    (* Table initialization: fTable_C *)
    fTable_C[0, 0] := 10.0000; fTable_C[0, 1] := -9999; fTable_C[0, 2] := 0.806885;
    fTable_C[1, 0] := 10.1617; fTable_C[1, 1] := -9999; fTable_C[1, 2] := 0.851522;
    fTable_C[2, 0] := 10.3261; fTable_C[2, 1] := -9999; fTable_C[2, 2] := 0.898628;
    fTable_C[3, 0] := 10.4931; fTable_C[3, 1] := -9999; fTable_C[3, 2] := 0.948341;
    fTable_C[4, 0] := 10.6628; fTable_C[4, 1] := -9999; fTable_C[4, 2] := 1.00080;
    fTable_C[5, 0] := 10.8353; fTable_C[5, 1] := -9999; fTable_C[5, 2] := 1.05755;
    fTable_C[6, 0] := 11.0106; fTable_C[6, 1] := -9999; fTable_C[6, 2] := 1.12167;
    fTable_C[7, 0] := 11.1886; fTable_C[7, 1] := -9999; fTable_C[7, 2] := 1.18968;
    fTable_C[8, 0] := 11.3696; fTable_C[8, 1] := -9999; fTable_C[8, 2] := 1.26181;
    fTable_C[9, 0] := 11.5535; fTable_C[9, 1] := -9999; fTable_C[9, 2] := 1.33832;
    fTable_C[10, 0] := 11.7404; fTable_C[10, 1] := -9999; fTable_C[10, 2] := 1.41946;
    fTable_C[11, 0] := 11.9303; fTable_C[11, 1] := -9999; fTable_C[11, 2] := 1.50553;
    fTable_C[12, 0] := 12.1232; fTable_C[12, 1] := -9999; fTable_C[12, 2] := 1.58971;
    fTable_C[13, 0] := 12.3193; fTable_C[13, 1] := -9999; fTable_C[13, 2] := 1.67820;
    fTable_C[14, 0] := 12.5186; fTable_C[14, 1] := -9999; fTable_C[14, 2] := 1.77161;
    fTable_C[15, 0] := 12.7210; fTable_C[15, 1] := -9999; fTable_C[15, 2] := 1.87023;
    fTable_C[16, 0] := 12.9268; fTable_C[16, 1] := -9999; fTable_C[16, 2] := 1.97433;
    fTable_C[17, 0] := 13.1359; fTable_C[17, 1] := -9999; fTable_C[17, 2] := 2.08423;
    fTable_C[18, 0] := 13.3483; fTable_C[18, 1] := -9999; fTable_C[18, 2] := 2.20025;
    fTable_C[19, 0] := 13.5642; fTable_C[19, 1] := -9999; fTable_C[19, 2] := 2.29235;
    fTable_C[20, 0] := 13.7836; fTable_C[20, 1] := -9999; fTable_C[20, 2] := 2.38287;
    fTable_C[21, 0] := 14.0066; fTable_C[21, 1] := -9999; fTable_C[21, 2] := 2.47696;
    fTable_C[22, 0] := 14.2331; fTable_C[22, 1] := -9999; fTable_C[22, 2] := 2.57477;
    fTable_C[23, 0] := 14.4633; fTable_C[23, 1] := -9999; fTable_C[23, 2] := 2.67645;
    fTable_C[24, 0] := 14.6973; fTable_C[24, 1] := -9999; fTable_C[24, 2] := 2.77114;
    fTable_C[25, 0] := 14.9350; fTable_C[25, 1] := -9999; fTable_C[25, 2] := 2.84605;
    fTable_C[26, 0] := 15.1765; fTable_C[26, 1] := -9999; fTable_C[26, 2] := 2.92298;
    fTable_C[27, 0] := 15.4220; fTable_C[27, 1] := -9999; fTable_C[27, 2] := 3.00199;
    fTable_C[28, 0] := 15.6714; fTable_C[28, 1] := -9999; fTable_C[28, 2] := 3.08313;
    fTable_C[29, 0] := 15.9249; fTable_C[29, 1] := -9999; fTable_C[29, 2] := 3.16647;
    fTable_C[30, 0] := 16.1825; fTable_C[30, 1] := -9999; fTable_C[30, 2] := 3.24213;
    fTable_C[31, 0] := 16.4442; fTable_C[31, 1] := -9999; fTable_C[31, 2] := 3.28778;
    fTable_C[32, 0] := 16.7102; fTable_C[32, 1] := -9999; fTable_C[32, 2] := 3.33408;
    fTable_C[33, 0] := 16.9805; fTable_C[33, 1] := -9999; fTable_C[33, 2] := 3.38103;
    fTable_C[34, 0] := 17.2551; fTable_C[34, 1] := -9999; fTable_C[34, 2] := 3.42863;
    fTable_C[35, 0] := 17.5342; fTable_C[35, 1] := -9999; fTable_C[35, 2] := 3.47691;
    fTable_C[36, 0] := 17.8178; fTable_C[36, 1] := -9999; fTable_C[36, 2] := 3.52041;
    fTable_C[37, 0] := 18.1060; fTable_C[37, 1] := -9999; fTable_C[37, 2] := 3.54277;
    fTable_C[38, 0] := 18.3989; fTable_C[38, 1] := -9999; fTable_C[38, 2] := 3.56528;
    fTable_C[39, 0] := 18.6964; fTable_C[39, 1] := -9999; fTable_C[39, 2] := 3.58793;
    fTable_C[40, 0] := 18.9988; fTable_C[40, 1] := -9999; fTable_C[40, 2] := 3.61072;
    fTable_C[41, 0] := 19.3061; fTable_C[41, 1] := -9999; fTable_C[41, 2] := 3.63366;
    fTable_C[42, 0] := 19.6184; fTable_C[42, 1] := -9999; fTable_C[42, 2] := 3.65674;
    fTable_C[43, 0] := 19.9357; fTable_C[43, 1] := -9999; fTable_C[43, 2] := 3.67997;
    fTable_C[44, 0] := 20.2582; fTable_C[44, 1] := -9999; fTable_C[44, 2] := 3.70335;
    fTable_C[45, 0] := 20.5858; fTable_C[45, 1] := -9999; fTable_C[45, 2] := 3.69489;
    fTable_C[46, 0] := 20.9188; fTable_C[46, 1] := -9999; fTable_C[46, 2] := 3.67204;
    fTable_C[47, 0] := 21.2571; fTable_C[47, 1] := -9999; fTable_C[47, 2] := 3.64934;
    fTable_C[48, 0] := 21.6009; fTable_C[48, 1] := -9999; fTable_C[48, 2] := 3.62677;
    fTable_C[49, 0] := 21.9503; fTable_C[49, 1] := -9999; fTable_C[49, 2] := 3.60434;
    fTable_C[50, 0] := 22.3053; fTable_C[50, 1] := -9999; fTable_C[50, 2] := 3.58205;
    fTable_C[51, 0] := 22.6661; fTable_C[51, 1] := -9999; fTable_C[51, 2] := 3.55990;
    fTable_C[52, 0] := 23.0327; fTable_C[52, 1] := -9999; fTable_C[52, 2] := 3.53320;
    fTable_C[53, 0] := 23.4053; fTable_C[53, 1] := -9999; fTable_C[53, 2] := 3.47892;
    fTable_C[54, 0] := 23.7838; fTable_C[54, 1] := -9999; fTable_C[54, 2] := 3.42547;
    fTable_C[55, 0] := 24.1685; fTable_C[55, 1] := -9999; fTable_C[55, 2] := 3.37285;
    fTable_C[56, 0] := 24.5594; fTable_C[56, 1] := -9999; fTable_C[56, 2] := 3.32103;
    fTable_C[57, 0] := 24.9566; fTable_C[57, 1] := -9999; fTable_C[57, 2] := 3.27000;
    fTable_C[58, 0] := 25.3603; fTable_C[58, 1] := -9999; fTable_C[58, 2] := 3.21977;
    fTable_C[59, 0] := 25.7705; fTable_C[59, 1] := -9999; fTable_C[59, 2] := 3.17030;
    fTable_C[60, 0] := 26.1873; fTable_C[60, 1] := -9999; fTable_C[60, 2] := 3.12096;
    fTable_C[61, 0] := 26.6109; fTable_C[61, 1] := -9999; fTable_C[61, 2] := 3.06350;
    fTable_C[62, 0] := 27.0413; fTable_C[62, 1] := -9999; fTable_C[62, 2] := 3.00708;
    fTable_C[63, 0] := 27.4786; fTable_C[63, 1] := -9999; fTable_C[63, 2] := 2.95171;
    fTable_C[64, 0] := 27.9231; fTable_C[64, 1] := -9999; fTable_C[64, 2] := 2.89736;
    fTable_C[65, 0] := 28.3747; fTable_C[65, 1] := -9999; fTable_C[65, 2] := 2.84401;
    fTable_C[66, 0] := 28.8337; fTable_C[66, 1] := -9999; fTable_C[66, 2] := 2.79164;
    fTable_C[67, 0] := 29.3000; fTable_C[67, 1] := 3.63318; fTable_C[67, 2] := 2.74024;
    fTable_C[68, 0] := 29.7739; fTable_C[68, 1] := 3.67378; fTable_C[68, 2] := 2.68978;
    fTable_C[69, 0] := 30.2555; fTable_C[69, 1] := 3.71270; fTable_C[69, 2] := 2.63618;
    fTable_C[70, 0] := 30.7449; fTable_C[70, 1] := 3.74753; fTable_C[70, 2] := 2.58360;
    fTable_C[71, 0] := 31.2421; fTable_C[71, 1] := 3.77973; fTable_C[71, 2] := 2.53206;
    fTable_C[72, 0] := 31.7475; fTable_C[72, 1] := 3.80969; fTable_C[72, 2] := 2.48155;
    fTable_C[73, 0] := 32.2609; fTable_C[73, 1] := 3.83764; fTable_C[73, 2] := 2.43205;
    fTable_C[74, 0] := 32.7827; fTable_C[74, 1] := 3.86374; fTable_C[74, 2] := 2.38354;
    fTable_C[75, 0] := 33.3130; fTable_C[75, 1] := 3.88807; fTable_C[75, 2] := 2.33599;
    fTable_C[76, 0] := 33.8518; fTable_C[76, 1] := 3.91071; fTable_C[76, 2] := 2.28940;
    fTable_C[77, 0] := 34.3993; fTable_C[77, 1] := 3.93156; fTable_C[77, 2] := 2.24373;
    fTable_C[78, 0] := 34.9557; fTable_C[78, 1] := 3.95026; fTable_C[78, 2] := 2.19898;
    fTable_C[79, 0] := 35.5211; fTable_C[79, 1] := 3.96709; fTable_C[79, 2] := 2.15799;
    fTable_C[80, 0] := 36.0956; fTable_C[80, 1] := 3.98488; fTable_C[80, 2] := 2.11827;
    fTable_C[81, 0] := 36.6794; fTable_C[81, 1] := 4.00253; fTable_C[81, 2] := 2.07928;
    fTable_C[82, 0] := 37.2727; fTable_C[82, 1] := 4.01992; fTable_C[82, 2] := 2.04101;
    fTable_C[83, 0] := 37.8755; fTable_C[83, 1] := 4.03712; fTable_C[83, 2] := 2.00344;
    fTable_C[84, 0] := 38.4882; fTable_C[84, 1] := 4.05432; fTable_C[84, 2] := 1.96657;
    fTable_C[85, 0] := 39.1107; fTable_C[85, 1] := 4.07360; fTable_C[85, 2] := 1.93037;
    fTable_C[86, 0] := 39.7432; fTable_C[86, 1] := 4.09449; fTable_C[86, 2] := 1.89011;
    fTable_C[87, 0] := 40.3861; fTable_C[87, 1] := 4.11010; fTable_C[87, 2] := 1.84650;
    fTable_C[88, 0] := 41.0393; fTable_C[88, 1] := 4.12229; fTable_C[88, 2] := 1.80390;
    fTable_C[89, 0] := 41.7031; fTable_C[89, 1] := 4.13211; fTable_C[89, 2] := 1.76228;
    fTable_C[90, 0] := 42.3776; fTable_C[90, 1] := 4.13985; fTable_C[90, 2] := 1.72163;
    fTable_C[91, 0] := 43.0630; fTable_C[91, 1] := 4.14559; fTable_C[91, 2] := 1.68191;
    fTable_C[92, 0] := 43.7595; fTable_C[92, 1] := 4.14925; fTable_C[92, 2] := 1.64310;
    fTable_C[93, 0] := 44.4673; fTable_C[93, 1] := 4.14955; fTable_C[93, 2] := 1.60520;
    fTable_C[94, 0] := 45.1865; fTable_C[94, 1] := 4.14584; fTable_C[94, 2] := 1.56917;
    fTable_C[95, 0] := 45.9174; fTable_C[95, 1] := 4.14175; fTable_C[95, 2] := 1.54376;
    fTable_C[96, 0] := 46.6600; fTable_C[96, 1] := 4.14174; fTable_C[96, 2] := 1.51876;
    fTable_C[97, 0] := 47.4147; fTable_C[97, 1] := 4.14300; fTable_C[97, 2] := 1.49417;
    fTable_C[98, 0] := 48.1816; fTable_C[98, 1] := 4.14486; fTable_C[98, 2] := 1.46998;
    fTable_C[99, 0] := 48.9609; fTable_C[99, 1] := 4.14698; fTable_C[99, 2] := 1.44618;
    fTable_C[100, 0] := 49.7528; fTable_C[100, 1] := 4.14913; fTable_C[100, 2] := 1.42276;
    fTable_C[101, 0] := 50.5576; fTable_C[101, 1] := 4.15113; fTable_C[101, 2] := 1.39972;
    fTable_C[102, 0] := 51.3753; fTable_C[102, 1] := 4.15277; fTable_C[102, 2] := 1.37705;
    fTable_C[103, 0] := 52.2062; fTable_C[103, 1] := 4.15371; fTable_C[103, 2] := 1.35475;
    fTable_C[104, 0] := 53.0506; fTable_C[104, 1] := 4.15307; fTable_C[104, 2] := 1.33282;
    fTable_C[105, 0] := 53.9087; fTable_C[105, 1] := 4.14960; fTable_C[105, 2] := 1.31546;
    fTable_C[106, 0] := 54.7806; fTable_C[106, 1] := 4.14997; fTable_C[106, 2] := 1.30168;
    fTable_C[107, 0] := 55.6667; fTable_C[107, 1] := 4.15270; fTable_C[107, 2] := 1.28804;
    fTable_C[108, 0] := 56.5670; fTable_C[108, 1] := 4.15681; fTable_C[108, 2] := 1.27454;
    fTable_C[109, 0] := 57.4820; fTable_C[109, 1] := 4.16209; fTable_C[109, 2] := 1.26118;
    fTable_C[110, 0] := 58.4117; fTable_C[110, 1] := 4.16851; fTable_C[110, 2] := 1.24797;
    fTable_C[111, 0] := 59.3564; fTable_C[111, 1] := 4.17625; fTable_C[111, 2] := 1.23489;
    fTable_C[112, 0] := 60.3165; fTable_C[112, 1] := 4.18600; fTable_C[112, 2] := 1.22195;
    fTable_C[113, 0] := 61.2921; fTable_C[113, 1] := 4.19949; fTable_C[113, 2] := 1.20654;
    fTable_C[114, 0] := 62.2834; fTable_C[114, 1] := 4.21096; fTable_C[114, 2] := 1.18498;
    fTable_C[115, 0] := 63.2908; fTable_C[115, 1] := 4.21910; fTable_C[115, 2] := 1.16381;
    fTable_C[116, 0] := 64.3145; fTable_C[116, 1] := 4.22582; fTable_C[116, 2] := 1.14301;
    fTable_C[117, 0] := 65.3547; fTable_C[117, 1] := 4.23161; fTable_C[117, 2] := 1.12258;
    fTable_C[118, 0] := 66.4118; fTable_C[118, 1] := 4.23666; fTable_C[118, 2] := 1.10252;
    fTable_C[119, 0] := 67.4859; fTable_C[119, 1] := 4.24111; fTable_C[119, 2] := 1.08282;
    fTable_C[120, 0] := 68.5775; fTable_C[120, 1] := 4.24504; fTable_C[120, 2] := 1.06347;
    fTable_C[121, 0] := 69.6867; fTable_C[121, 1] := 4.24852; fTable_C[121, 2] := 1.04447;
    fTable_C[122, 0] := 70.8138; fTable_C[122, 1] := 4.25160; fTable_C[122, 2] := 1.02580;
    fTable_C[123, 0] := 71.9591; fTable_C[123, 1] := 4.25430; fTable_C[123, 2] := 1.00747;
    fTable_C[124, 0] := 73.1230; fTable_C[124, 1] := 4.25667; fTable_C[124, 2] := 0.989470;
    fTable_C[125, 0] := 74.3057; fTable_C[125, 1] := 4.25872; fTable_C[125, 2] := 0.971788;
    fTable_C[126, 0] := 75.5076; fTable_C[126, 1] := 4.26047; fTable_C[126, 2] := 0.954423;
    fTable_C[127, 0] := 76.7289; fTable_C[127, 1] := 4.26194; fTable_C[127, 2] := 0.937369;
    fTable_C[128, 0] := 77.9699; fTable_C[128, 1] := 4.26314; fTable_C[128, 2] := 0.920617;
    fTable_C[129, 0] := 79.2310; fTable_C[129, 1] := 4.26408; fTable_C[129, 2] := 0.904167;
    fTable_C[130, 0] := 80.5125; fTable_C[130, 1] := 4.26478; fTable_C[130, 2] := 0.888009;
    fTable_C[131, 0] := 81.8147; fTable_C[131, 1] := 4.26524; fTable_C[131, 2] := 0.872141;
    fTable_C[132, 0] := 83.1380; fTable_C[132, 1] := 4.26546; fTable_C[132, 2] := 0.856556;
    fTable_C[133, 0] := 84.4827; fTable_C[133, 1] := 4.26547; fTable_C[133, 2] := 0.841250;
    fTable_C[134, 0] := 85.8491; fTable_C[134, 1] := 4.26525; fTable_C[134, 2] := 0.826217;
    fTable_C[135, 0] := 87.2377; fTable_C[135, 1] := 4.26481; fTable_C[135, 2] := 0.811453;
    fTable_C[136, 0] := 88.6487; fTable_C[136, 1] := 4.26417; fTable_C[136, 2] := 0.796952;
    fTable_C[137, 0] := 90.0825; fTable_C[137, 1] := 4.26332; fTable_C[137, 2] := 0.782711;
    fTable_C[138, 0] := 91.5395; fTable_C[138, 1] := 4.26226; fTable_C[138, 2] := 0.768724;
    fTable_C[139, 0] := 93.0201; fTable_C[139, 1] := 4.26100; fTable_C[139, 2] := 0.754987;
    fTable_C[140, 0] := 94.5246; fTable_C[140, 1] := 4.25953; fTable_C[140, 2] := 0.741496;
    fTable_C[141, 0] := 96.0535; fTable_C[141, 1] := 4.25787; fTable_C[141, 2] := 0.728246;
    fTable_C[142, 0] := 97.6071; fTable_C[142, 1] := 4.25600; fTable_C[142, 2] := 0.715232;
    fTable_C[143, 0] := 99.1858; fTable_C[143, 1] := 4.25393; fTable_C[143, 2] := 0.702451;
    fTable_C[144, 0] := 100.790; fTable_C[144, 1] := 4.25166; fTable_C[144, 2] := 0.689898;
    fTable_C[145, 0] := 102.420; fTable_C[145, 1] := 4.24919; fTable_C[145, 2] := 0.677570;
    fTable_C[146, 0] := 104.077; fTable_C[146, 1] := 4.24651; fTable_C[146, 2] := 0.665462;
    fTable_C[147, 0] := 105.760; fTable_C[147, 1] := 4.24363; fTable_C[147, 2] := 0.653570;
    fTable_C[148, 0] := 107.471; fTable_C[148, 1] := 4.24054; fTable_C[148, 2] := 0.641891;
    fTable_C[149, 0] := 109.209; fTable_C[149, 1] := 4.23724; fTable_C[149, 2] := 0.630421;
    fTable_C[150, 0] := 110.975; fTable_C[150, 1] := 4.23373; fTable_C[150, 2] := 0.619156;
    fTable_C[151, 0] := 112.770; fTable_C[151, 1] := 4.23000; fTable_C[151, 2] := 0.608091;
    fTable_C[152, 0] := 114.594; fTable_C[152, 1] := 4.22606; fTable_C[152, 2] := 0.597224;
    fTable_C[153, 0] := 116.448; fTable_C[153, 1] := 4.22189; fTable_C[153, 2] := 0.586552;
    fTable_C[154, 0] := 118.331; fTable_C[154, 1] := 4.21751; fTable_C[154, 2] := 0.576071;
    fTable_C[155, 0] := 120.245; fTable_C[155, 1] := 4.21289; fTable_C[155, 2] := 0.565777;
    fTable_C[156, 0] := 122.190; fTable_C[156, 1] := 4.20806; fTable_C[156, 2] := 0.555666;
    fTable_C[157, 0] := 124.166; fTable_C[157, 1] := 4.20299; fTable_C[157, 2] := 0.545737;
    fTable_C[158, 0] := 126.175; fTable_C[158, 1] := 4.19772; fTable_C[158, 2] := 0.535985;
    fTable_C[159, 0] := 128.215; fTable_C[159, 1] := 4.19225; fTable_C[159, 2] := 0.526406;
    fTable_C[160, 0] := 130.289; fTable_C[160, 1] := 4.18666; fTable_C[160, 2] := 0.517000;
    fTable_C[161, 0] := 132.397; fTable_C[161, 1] := 4.18122; fTable_C[161, 2] := 0.507761;
    fTable_C[162, 0] := 134.538; fTable_C[162, 1] := 4.17533; fTable_C[162, 2] := 0.497457;
    fTable_C[163, 0] := 136.714; fTable_C[163, 1] := 4.16860; fTable_C[163, 2] := 0.487361;
    fTable_C[164, 0] := 138.925; fTable_C[164, 1] := 4.16122; fTable_C[164, 2] := 0.477469;
    fTable_C[165, 0] := 141.172; fTable_C[165, 1] := 4.15329; fTable_C[165, 2] := 0.467777;
    fTable_C[166, 0] := 143.456; fTable_C[166, 1] := 4.14484; fTable_C[166, 2] := 0.458283;
    fTable_C[167, 0] := 145.776; fTable_C[167, 1] := 4.13587; fTable_C[167, 2] := 0.448981;
    fTable_C[168, 0] := 148.134; fTable_C[168, 1] := 4.12638; fTable_C[168, 2] := 0.439868;
    fTable_C[169, 0] := 150.530; fTable_C[169, 1] := 4.11636; fTable_C[169, 2] := 0.430941;
    fTable_C[170, 0] := 152.964; fTable_C[170, 1] := 4.10578; fTable_C[170, 2] := 0.422193;
    fTable_C[171, 0] := 155.439; fTable_C[171, 1] := 4.09464; fTable_C[171, 2] := 0.413624;
    fTable_C[172, 0] := 157.953; fTable_C[172, 1] := 4.08290; fTable_C[172, 2] := 0.405229;
    fTable_C[173, 0] := 160.507; fTable_C[173, 1] := 4.07054; fTable_C[173, 2] := 0.397004;
    fTable_C[174, 0] := 163.103; fTable_C[174, 1] := 4.05754; fTable_C[174, 2] := 0.388946;
    fTable_C[175, 0] := 165.742; fTable_C[175, 1] := 4.04385; fTable_C[175, 2] := 0.381052;
    fTable_C[176, 0] := 168.422; fTable_C[176, 1] := 4.02945; fTable_C[176, 2] := 0.373318;
    fTable_C[177, 0] := 171.146; fTable_C[177, 1] := 4.01429; fTable_C[177, 2] := 0.365741;
    fTable_C[178, 0] := 173.915; fTable_C[178, 1] := 3.99834; fTable_C[178, 2] := 0.358317;
    fTable_C[179, 0] := 176.727; fTable_C[179, 1] := 3.98158; fTable_C[179, 2] := 0.351045;
    fTable_C[180, 0] := 179.586; fTable_C[180, 1] := 3.96398; fTable_C[180, 2] := 0.343919;
    fTable_C[181, 0] := 182.491; fTable_C[181, 1] := 3.94558; fTable_C[181, 2] := 0.336939;
    fTable_C[182, 0] := 185.442; fTable_C[182, 1] := 3.92716; fTable_C[182, 2] := 0.330100;
    fTable_C[183, 0] := 188.442; fTable_C[183, 1] := 3.90705; fTable_C[183, 2] := 0.320995;
    fTable_C[184, 0] := 191.489; fTable_C[184, 1] := 3.88443; fTable_C[184, 2] := 0.312096;
    fTable_C[185, 0] := 194.587; fTable_C[185, 1] := 3.85977; fTable_C[185, 2] := 0.303443;
    fTable_C[186, 0] := 197.734; fTable_C[186, 1] := 3.83308; fTable_C[186, 2] := 0.295031;
    fTable_C[187, 0] := 200.932; fTable_C[187, 1] := 3.80428; fTable_C[187, 2] := 0.286851;
    fTable_C[188, 0] := 204.182; fTable_C[188, 1] := 3.77323; fTable_C[188, 2] := 0.278898;
    fTable_C[189, 0] := 207.485; fTable_C[189, 1] := 3.73972; fTable_C[189, 2] := 0.271166;
    fTable_C[190, 0] := 210.840; fTable_C[190, 1] := 3.70351; fTable_C[190, 2] := 0.263648;
    fTable_C[191, 0] := 214.251; fTable_C[191, 1] := 3.66428; fTable_C[191, 2] := 0.256338;
    fTable_C[192, 0] := 217.716; fTable_C[192, 1] := 3.62164; fTable_C[192, 2] := 0.249231;
    fTable_C[193, 0] := 221.237; fTable_C[193, 1] := 3.57499; fTable_C[193, 2] := 0.242516;
    fTable_C[194, 0] := 224.816; fTable_C[194, 1] := 3.52435; fTable_C[194, 2] := 0.236381;
    fTable_C[195, 0] := 228.452; fTable_C[195, 1] := 3.46902; fTable_C[195, 2] := 0.230402;
    fTable_C[196, 0] := 232.147; fTable_C[196, 1] := 3.40812; fTable_C[196, 2] := 0.224573;
    fTable_C[197, 0] := 235.902; fTable_C[197, 1] := 3.34061; fTable_C[197, 2] := 0.218892;
    fTable_C[198, 0] := 239.717; fTable_C[198, 1] := 3.26522; fTable_C[198, 2] := 0.213355;
    fTable_C[199, 0] := 243.595; fTable_C[199, 1] := 3.18027; fTable_C[199, 2] := 0.207958;
    fTable_C[200, 0] := 247.535; fTable_C[200, 1] := 3.08474; fTable_C[200, 2] := 0.202179;
    fTable_C[201, 0] := 251.538; fTable_C[201, 1] := 2.97293; fTable_C[201, 2] := 0.194683;
    fTable_C[202, 0] := 255.607; fTable_C[202, 1] := 2.84002; fTable_C[202, 2] := 0.187465;
    fTable_C[203, 0] := 259.741; fTable_C[203, 1] := 2.67985; fTable_C[203, 2] := 0.180514;
    fTable_C[204, 0] := 263.942; fTable_C[204, 1] := 2.48138; fTable_C[204, 2] := 0.173821;
    fTable_C[205, 0] := 268.211; fTable_C[205, 1] := 2.22505; fTable_C[205, 2] := 0.167377;
    fTable_C[206, 0] := 272.549; fTable_C[206, 1] := 1.87159; fTable_C[206, 2] := 0.161171;
    fTable_C[207, 0] := 276.957; fTable_C[207, 1] := 1.32192; fTable_C[207, 2] := 0.155195;
    fTable_C[208, 0] := 281.437; fTable_C[208, 1] := 0.158573; fTable_C[208, 2] := 0.149441;
    fTable_C[209, 0] := 284.100; fTable_C[209, 1] := -4.04882; fTable_C[209, 2] := 0.146163;
    fTable_C[210, 0] := 284.300; fTable_C[210, 1] := -4.04031; fTable_C[210, 2] := 4.18872;
    fTable_C[211, 0] := 285.989; fTable_C[211, 1] := -0.283330; fTable_C[211, 2] := 4.15857;
    fTable_C[212, 0] := 290.615; fTable_C[212, 1] := 1.43967; fTable_C[212, 2] := 4.07798;
    fTable_C[213, 0] := 295.315; fTable_C[213, 1] := 2.20576; fTable_C[213, 2] := 3.99896;
    fTable_C[214, 0] := 300.092; fTable_C[214, 1] := 2.71286; fTable_C[214, 2] := 3.92146;
    fTable_C[215, 0] := 304.945; fTable_C[215, 1] := 3.09475; fTable_C[215, 2] := 3.84546;
    fTable_C[216, 0] := 309.878; fTable_C[216, 1] := 3.40186; fTable_C[216, 2] := 3.77095;
    fTable_C[217, 0] := 314.890; fTable_C[217, 1] := 3.65884; fTable_C[217, 2] := 3.69787;
    fTable_C[218, 0] := 319.983; fTable_C[218, 1] := 3.87969; fTable_C[218, 2] := 3.62620;
    fTable_C[219, 0] := 325.158; fTable_C[219, 1] := 4.07315; fTable_C[219, 2] := 3.55593;
    fTable_C[220, 0] := 330.418; fTable_C[220, 1] := 4.24510; fTable_C[220, 2] := 3.48703;
    fTable_C[221, 0] := 335.762; fTable_C[221, 1] := 4.39967; fTable_C[221, 2] := 3.41945;
    fTable_C[222, 0] := 341.192; fTable_C[222, 1] := 4.53993; fTable_C[222, 2] := 3.35318;
    fTable_C[223, 0] := 346.711; fTable_C[223, 1] := 4.66823; fTable_C[223, 2] := 3.28820;
    fTable_C[224, 0] := 352.319; fTable_C[224, 1] := 4.78642; fTable_C[224, 2] := 3.22448;
    fTable_C[225, 0] := 358.017; fTable_C[225, 1] := 4.89606; fTable_C[225, 2] := 3.16200;
    fTable_C[226, 0] := 363.808; fTable_C[226, 1] := 4.99852; fTable_C[226, 2] := 3.10072;
    fTable_C[227, 0] := 369.692; fTable_C[227, 1] := 5.09524; fTable_C[227, 2] := 3.04063;
    fTable_C[228, 0] := 375.672; fTable_C[228, 1] := 5.18910; fTable_C[228, 2] := 2.98170;
    fTable_C[229, 0] := 381.748; fTable_C[229, 1] := 5.27926; fTable_C[229, 2] := 2.91649;
    fTable_C[230, 0] := 387.922; fTable_C[230, 1] := 5.36049; fTable_C[230, 2] := 2.84817;
    fTable_C[231, 0] := 394.197; fTable_C[231, 1] := 5.43267; fTable_C[231, 2] := 2.78144;
    fTable_C[232, 0] := 400.573; fTable_C[232, 1] := 5.49897; fTable_C[232, 2] := 2.71628;
    fTable_C[233, 0] := 407.052; fTable_C[233, 1] := 5.56010; fTable_C[233, 2] := 2.65264;
    fTable_C[234, 0] := 413.635; fTable_C[234, 1] := 5.61669; fTable_C[234, 2] := 2.59050;
    fTable_C[235, 0] := 420.326; fTable_C[235, 1] := 5.66920; fTable_C[235, 2] := 2.52981;
    fTable_C[236, 0] := 427.124; fTable_C[236, 1] := 5.71803; fTable_C[236, 2] := 2.47054;
    fTable_C[237, 0] := 434.032; fTable_C[237, 1] := 5.76351; fTable_C[237, 2] := 2.41266;
    fTable_C[238, 0] := 441.052; fTable_C[238, 1] := 5.80593; fTable_C[238, 2] := 2.35614;
    fTable_C[239, 0] := 448.186; fTable_C[239, 1] := 5.84557; fTable_C[239, 2] := 2.30094;
    fTable_C[240, 0] := 455.435; fTable_C[240, 1] := 5.88264; fTable_C[240, 2] := 2.24703;
    fTable_C[241, 0] := 462.802; fTable_C[241, 1] := 5.91737; fTable_C[241, 2] := 2.19439;
    fTable_C[242, 0] := 470.287; fTable_C[242, 1] := 5.94998; fTable_C[242, 2] := 2.14298;
    fTable_C[243, 0] := 477.894; fTable_C[243, 1] := 5.98074; fTable_C[243, 2] := 2.09278;
    fTable_C[244, 0] := 485.623; fTable_C[244, 1] := 6.01022; fTable_C[244, 2] := 2.04367;
    fTable_C[245, 0] := 493.478; fTable_C[245, 1] := 6.03767; fTable_C[245, 2] := 1.99418;
    fTable_C[246, 0] := 501.459; fTable_C[246, 1] := 6.06268; fTable_C[246, 2] := 1.94589;
    fTable_C[247, 0] := 509.570; fTable_C[247, 1] := 6.08579; fTable_C[247, 2] := 1.89876;
    fTable_C[248, 0] := 517.812; fTable_C[248, 1] := 6.10721; fTable_C[248, 2] := 1.85278;
    fTable_C[249, 0] := 526.187; fTable_C[249, 1] := 6.12709; fTable_C[249, 2] := 1.80791;
    fTable_C[250, 0] := 534.698; fTable_C[250, 1] := 6.14556; fTable_C[250, 2] := 1.76412;
    fTable_C[251, 0] := 543.346; fTable_C[251, 1] := 6.16271; fTable_C[251, 2] := 1.72140;
    fTable_C[252, 0] := 552.134; fTable_C[252, 1] := 6.17864; fTable_C[252, 2] := 1.67971;
    fTable_C[253, 0] := 561.065; fTable_C[253, 1] := 6.19344; fTable_C[253, 2] := 1.63903;
    fTable_C[254, 0] := 570.139; fTable_C[254, 1] := 6.20717; fTable_C[254, 2] := 1.59933;
    fTable_C[255, 0] := 579.361; fTable_C[255, 1] := 6.21992; fTable_C[255, 2] := 1.56060;
    fTable_C[256, 0] := 588.732; fTable_C[256, 1] := 6.23174; fTable_C[256, 2] := 1.52281;
    fTable_C[257, 0] := 598.254; fTable_C[257, 1] := 6.24271; fTable_C[257, 2] := 1.48593;
    fTable_C[258, 0] := 607.930; fTable_C[258, 1] := 6.25287; fTable_C[258, 2] := 1.44994;
    fTable_C[259, 0] := 617.763; fTable_C[259, 1] := 6.26227; fTable_C[259, 2] := 1.41483;
    fTable_C[260, 0] := 627.755; fTable_C[260, 1] := 6.27097; fTable_C[260, 2] := 1.38056;
    fTable_C[261, 0] := 637.908; fTable_C[261, 1] := 6.27900; fTable_C[261, 2] := 1.34713;
    fTable_C[262, 0] := 648.226; fTable_C[262, 1] := 6.28639; fTable_C[262, 2] := 1.31450;
    fTable_C[263, 0] := 658.711; fTable_C[263, 1] := 6.29312; fTable_C[263, 2] := 1.28267;
    fTable_C[264, 0] := 669.365; fTable_C[264, 1] := 6.29901; fTable_C[264, 2] := 1.25160;
    fTable_C[265, 0] := 680.191; fTable_C[265, 1] := 6.30406; fTable_C[265, 2] := 1.22249;
    fTable_C[266, 0] := 691.193; fTable_C[266, 1] := 6.30972; fTable_C[266, 2] := 1.19523;
    fTable_C[267, 0] := 702.372; fTable_C[267, 1] := 6.31822; fTable_C[267, 2] := 1.16897;
    fTable_C[268, 0] := 713.733; fTable_C[268, 1] := 6.32783; fTable_C[268, 2] := 1.13958;
    fTable_C[269, 0] := 725.277; fTable_C[269, 1] := 6.33449; fTable_C[269, 2] := 1.10844;
    fTable_C[270, 0] := 737.008; fTable_C[270, 1] := 6.33933; fTable_C[270, 2] := 1.07816;
    fTable_C[271, 0] := 748.928; fTable_C[271, 1] := 6.34306; fTable_C[271, 2] := 1.04871;
    fTable_C[272, 0] := 761.042; fTable_C[272, 1] := 6.34594; fTable_C[272, 2] := 1.02006;
    fTable_C[273, 0] := 773.351; fTable_C[273, 1] := 6.34813; fTable_C[273, 2] := 0.992182;
    fTable_C[274, 0] := 785.859; fTable_C[274, 1] := 6.34973; fTable_C[274, 2] := 0.965046;
    fTable_C[275, 0] := 798.570; fTable_C[275, 1] := 6.35080; fTable_C[275, 2] := 0.938635;
    fTable_C[276, 0] := 811.486; fTable_C[276, 1] := 6.35140; fTable_C[276, 2] := 0.912939;
    fTable_C[277, 0] := 824.611; fTable_C[277, 1] := 6.35160; fTable_C[277, 2] := 0.887954;
    fTable_C[278, 0] := 837.949; fTable_C[278, 1] := 6.35148; fTable_C[278, 2] := 0.863661;
    fTable_C[279, 0] := 851.502; fTable_C[279, 1] := 6.35111; fTable_C[279, 2] := 0.839923;
    fTable_C[280, 0] := 865.274; fTable_C[280, 1] := 6.35042; fTable_C[280, 2] := 0.816714;
    fTable_C[281, 0] := 879.269; fTable_C[281, 1] := 6.34934; fTable_C[281, 2] := 0.794041;
    fTable_C[282, 0] := 893.491; fTable_C[282, 1] := 6.34793; fTable_C[282, 2] := 0.772006;
    fTable_C[283, 0] := 907.943; fTable_C[283, 1] := 6.34628; fTable_C[283, 2] := 0.750584;
    fTable_C[284, 0] := 922.628; fTable_C[284, 1] := 6.34445; fTable_C[284, 2] := 0.729761;
    fTable_C[285, 0] := 937.551; fTable_C[285, 1] := 6.34244; fTable_C[285, 2] := 0.709358;
    fTable_C[286, 0] := 952.715; fTable_C[286, 1] := 6.34016; fTable_C[286, 2] := 0.689500;
    fTable_C[287, 0] := 968.124; fTable_C[287, 1] := 6.33768; fTable_C[287, 2] := 0.670177;
    fTable_C[288, 0] := 983.783; fTable_C[288, 1] := 6.33503; fTable_C[288, 2] := 0.651378;
    fTable_C[289, 0] := 999.695; fTable_C[289, 1] := 6.33222; fTable_C[289, 2] := 0.633116;
    fTable_C[290, 0] := 1015.86; fTable_C[290, 1] := 6.32930; fTable_C[290, 2] := 0.615377;
    fTable_C[291, 0] := 1032.29; fTable_C[291, 1] := 6.32643; fTable_C[291, 2] := 0.598194;
    fTable_C[292, 0] := 1048.99; fTable_C[292, 1] := 6.32362; fTable_C[292, 2] := 0.581226;
    fTable_C[293, 0] := 1065.96; fTable_C[293, 1] := 6.32048; fTable_C[293, 2] := 0.564459;
    fTable_C[294, 0] := 1083.20; fTable_C[294, 1] := 6.31710; fTable_C[294, 2] := 0.548198;
    fTable_C[295, 0] := 1100.72; fTable_C[295, 1] := 6.31359; fTable_C[295, 2] := 0.532391;
    fTable_C[296, 0] := 1118.52; fTable_C[296, 1] := 6.30996; fTable_C[296, 2] := 0.517020;
    fTable_C[297, 0] := 1136.61; fTable_C[297, 1] := 6.30622; fTable_C[297, 2] := 0.502116;
    fTable_C[298, 0] := 1155; fTable_C[298, 1] := 6.30242; fTable_C[298, 2] := 0.487640;
    fTable_C[299, 0] := 1173.68; fTable_C[299, 1] := 6.29857; fTable_C[299, 2] := 0.473579;
    fTable_C[300, 0] := 1192.66; fTable_C[300, 1] := 6.29469; fTable_C[300, 2] := 0.459933;
    fTable_C[301, 0] := 1211.95; fTable_C[301, 1] := 6.29081; fTable_C[301, 2] := 0.446675;
    fTable_C[302, 0] := 1231.55; fTable_C[302, 1] := 6.28694; fTable_C[302, 2] := 0.433794;
    fTable_C[303, 0] := 1251.47; fTable_C[303, 1] := 6.28313; fTable_C[303, 2] := 0.421175;
    fTable_C[304, 0] := 1271.72; fTable_C[304, 1] := 6.27931; fTable_C[304, 2] := 0.408804;
    fTable_C[305, 0] := 1292.29; fTable_C[305, 1] := 6.27534; fTable_C[305, 2] := 0.396652;
    fTable_C[306, 0] := 1313.19; fTable_C[306, 1] := 6.27127; fTable_C[306, 2] := 0.384872;
    fTable_C[307, 0] := 1334.43; fTable_C[307, 1] := 6.26716; fTable_C[307, 2] := 0.373439;
    fTable_C[308, 0] := 1356.01; fTable_C[308, 1] := 6.26302; fTable_C[308, 2] := 0.362342;
    fTable_C[309, 0] := 1377.94; fTable_C[309, 1] := 6.25886; fTable_C[309, 2] := 0.351578;
    fTable_C[310, 0] := 1400.23; fTable_C[310, 1] := 6.25469; fTable_C[310, 2] := 0.341132;
    fTable_C[311, 0] := 1422.88; fTable_C[311, 1] := 6.25054; fTable_C[311, 2] := 0.330994;
    fTable_C[312, 0] := 1445.89; fTable_C[312, 1] := 6.24640; fTable_C[312, 2] := 0.321159;
    fTable_C[313, 0] := 1469.28; fTable_C[313, 1] := 6.24230; fTable_C[313, 2] := 0.311605;
    fTable_C[314, 0] := 1493.04; fTable_C[314, 1] := 6.23822; fTable_C[314, 2] := 0.302316;
    fTable_C[315, 0] := 1517.19; fTable_C[315, 1] := 6.23418; fTable_C[315, 2] := 0.293230;
    fTable_C[316, 0] := 1541.73; fTable_C[316, 1] := 6.23010; fTable_C[316, 2] := 0.284407;
    fTable_C[317, 0] := 1566.67; fTable_C[317, 1] := 6.22604; fTable_C[317, 2] := 0.275847;
    fTable_C[318, 0] := 1592.01; fTable_C[318, 1] := 6.22200; fTable_C[318, 2] := 0.267545;
    fTable_C[319, 0] := 1617.76; fTable_C[319, 1] := 6.21798; fTable_C[319, 2] := 0.259493;
    fTable_C[320, 0] := 1643.92; fTable_C[320, 1] := 6.21400; fTable_C[320, 2] := 0.251684;
    fTable_C[321, 0] := 1670.51; fTable_C[321, 1] := 6.21005; fTable_C[321, 2] := 0.244110;
    fTable_C[322, 0] := 1697.53; fTable_C[322, 1] := 6.20616; fTable_C[322, 2] := 0.236764;
    fTable_C[323, 0] := 1724.99; fTable_C[323, 1] := 6.20233; fTable_C[323, 2] := 0.229642;
    fTable_C[324, 0] := 1752.89; fTable_C[324, 1] := 6.19857; fTable_C[324, 2] := 0.222665;
    fTable_C[325, 0] := 1781.24; fTable_C[325, 1] := 6.19480; fTable_C[325, 2] := 0.215877;
    fTable_C[326, 0] := 1810.05; fTable_C[326, 1] := 6.19106; fTable_C[326, 2] := 0.209279;
    fTable_C[327, 0] := 1839.32; fTable_C[327, 1] := 6.18734; fTable_C[327, 2] := 0.202884;
    fTable_C[328, 0] := 1869.07; fTable_C[328, 1] := 6.18366; fTable_C[328, 2] := 0.196685;
    fTable_C[329, 0] := 1899.30; fTable_C[329, 1] := 6.18003; fTable_C[329, 2] := 0.190676;
    fTable_C[330, 0] := 1930.02; fTable_C[330, 1] := 6.17643; fTable_C[330, 2] := 0.184850;
    fTable_C[331, 0] := 1961.24; fTable_C[331, 1] := 6.17288; fTable_C[331, 2] := 0.179202;
    fTable_C[332, 0] := 1992.96; fTable_C[332, 1] := 6.16938; fTable_C[332, 2] := 0.173726;
    fTable_C[333, 0] := 2025.20; fTable_C[333, 1] := 6.16594; fTable_C[333, 2] := 0.168474;
    fTable_C[334, 0] := 2057.95; fTable_C[334, 1] := 6.16261; fTable_C[334, 2] := 0.163292;
    fTable_C[335, 0] := 2091.24; fTable_C[335, 1] := 6.15928; fTable_C[335, 2] := 0.158263;
    fTable_C[336, 0] := 2125.06; fTable_C[336, 1] := 6.15600; fTable_C[336, 2] := 0.153384;
    fTable_C[337, 0] := 2159.43; fTable_C[337, 1] := 6.15276; fTable_C[337, 2] := 0.148648;
    fTable_C[338, 0] := 2194.36; fTable_C[338, 1] := 6.14957; fTable_C[338, 2] := 0.144053;
    fTable_C[339, 0] := 2229.85; fTable_C[339, 1] := 6.14643; fTable_C[339, 2] := 0.139593;
    fTable_C[340, 0] := 2265.92; fTable_C[340, 1] := 6.14334; fTable_C[340, 2] := 0.135267;
    fTable_C[341, 0] := 2302.57; fTable_C[341, 1] := 6.14028; fTable_C[341, 2] := 0.131069;
    fTable_C[342, 0] := 2339.81; fTable_C[342, 1] := 6.13729; fTable_C[342, 2] := 0.126998;
    fTable_C[343, 0] := 2377.66; fTable_C[343, 1] := 6.13433; fTable_C[343, 2] := 0.123042;
    fTable_C[344, 0] := 2416.11; fTable_C[344, 1] := 6.13143; fTable_C[344, 2] := 0.119210;
    fTable_C[345, 0] := 2455.19; fTable_C[345, 1] := 6.12857; fTable_C[345, 2] := 0.115492;
    fTable_C[346, 0] := 2494.90; fTable_C[346, 1] := 6.12576; fTable_C[346, 2] := 0.111882;
    fTable_C[347, 0] := 2535.26; fTable_C[347, 1] := 6.12300; fTable_C[347, 2] := 0.108383;
    fTable_C[348, 0] := 2576.26; fTable_C[348, 1] := 6.12028; fTable_C[348, 2] := 0.104990;
    fTable_C[349, 0] := 2617.93; fTable_C[349, 1] := 6.11762; fTable_C[349, 2] := 0.101694;
    fTable_C[350, 0] := 2660.27; fTable_C[350, 1] := 6.11500; fTable_C[350, 2] := 0.0985042;
    fTable_C[351, 0] := 2703.30; fTable_C[351, 1] := 6.11243; fTable_C[351, 2] := 0.0954028;
    fTable_C[352, 0] := 2747.03; fTable_C[352, 1] := 6.10990; fTable_C[352, 2] := 0.0923971;
    fTable_C[353, 0] := 2791.46; fTable_C[353, 1] := 6.10742; fTable_C[353, 2] := 0.0894832;
    fTable_C[354, 0] := 2836.61; fTable_C[354, 1] := 6.10498; fTable_C[354, 2] := 0.0866617;
    fTable_C[355, 0] := 2882.49; fTable_C[355, 1] := 6.10259; fTable_C[355, 2] := 0.0839148;
    fTable_C[356, 0] := 2929.11; fTable_C[356, 1] := 6.10024; fTable_C[356, 2] := 0.0812599;
    fTable_C[357, 0] := 2976.48; fTable_C[357, 1] := 6.09794; fTable_C[357, 2] := 0.0786821;
    fTable_C[358, 0] := 3024.63; fTable_C[358, 1] := 6.09569; fTable_C[358, 2] := 0.0761825;
    fTable_C[359, 0] := 3073.55; fTable_C[359, 1] := 6.09347; fTable_C[359, 2] := 0.0737584;
    fTable_C[360, 0] := 3123.26; fTable_C[360, 1] := 6.09130; fTable_C[360, 2] := 0.0714080;
    fTable_C[361, 0] := 3173.78; fTable_C[361, 1] := 6.08917; fTable_C[361, 2] := 0.0691288;
    fTable_C[362, 0] := 3225.11; fTable_C[362, 1] := 6.08708; fTable_C[362, 2] := 0.0669194;
    fTable_C[363, 0] := 3277.27; fTable_C[363, 1] := 6.08503; fTable_C[363, 2] := 0.0647767;
    fTable_C[364, 0] := 3330.28; fTable_C[364, 1] := 6.08302; fTable_C[364, 2] := 0.0626991;
    fTable_C[365, 0] := 3384.15; fTable_C[365, 1] := 6.08105; fTable_C[365, 2] := 0.0606853;
    fTable_C[366, 0] := 3438.88; fTable_C[366, 1] := 6.07912; fTable_C[366, 2] := 0.0587327;
    fTable_C[367, 0] := 3494.50; fTable_C[367, 1] := 6.07723; fTable_C[367, 2] := 0.0568396;
    fTable_C[368, 0] := 3551.02; fTable_C[368, 1] := 6.07538; fTable_C[368, 2] := 0.0550042;
    fTable_C[369, 0] := 3608.46; fTable_C[369, 1] := 6.07357; fTable_C[369, 2] := 0.0532244;
    fTable_C[370, 0] := 3666.82; fTable_C[370, 1] := 6.07179; fTable_C[370, 2] := 0.0514997;
    fTable_C[371, 0] := 3726.13; fTable_C[371, 1] := 6.07005; fTable_C[371, 2] := 0.0498278;
    fTable_C[372, 0] := 3786.40; fTable_C[372, 1] := 6.06834; fTable_C[372, 2] := 0.0482071;
    fTable_C[373, 0] := 3847.64; fTable_C[373, 1] := 6.06667; fTable_C[373, 2] := 0.0466352;
    fTable_C[374, 0] := 3909.87; fTable_C[374, 1] := 6.06504; fTable_C[374, 2] := 0.0451127;
    fTable_C[375, 0] := 3973.11; fTable_C[375, 1] := 6.06343; fTable_C[375, 2] := 0.0436367;
    fTable_C[376, 0] := 4037.38; fTable_C[376, 1] := 6.06186; fTable_C[376, 2] := 0.0422212;
    fTable_C[377, 0] := 4102.68; fTable_C[377, 1] := 6.06033; fTable_C[377, 2] := 0.0408351;
    fTable_C[378, 0] := 4169.03; fTable_C[378, 1] := 6.05883; fTable_C[378, 2] := 0.0394919;
    fTable_C[379, 0] := 4236.46; fTable_C[379, 1] := 6.05736; fTable_C[379, 2] := 0.0381921;
    fTable_C[380, 0] := 4304.98; fTable_C[380, 1] := 6.05592; fTable_C[380, 2] := 0.0369324;
    fTable_C[381, 0] := 4374.62; fTable_C[381, 1] := 6.05451; fTable_C[381, 2] := 0.0357130;
    fTable_C[382, 0] := 4445.37; fTable_C[382, 1] := 6.05313; fTable_C[382, 2] := 0.0345329;
    fTable_C[383, 0] := 4517.27; fTable_C[383, 1] := 6.05178; fTable_C[383, 2] := 0.0333896;
    fTable_C[384, 0] := 4590.33; fTable_C[384, 1] := 6.05046; fTable_C[384, 2] := 0.0322825;
    fTable_C[385, 0] := 4664.58; fTable_C[385, 1] := 6.04917; fTable_C[385, 2] := 0.0312100;
    fTable_C[386, 0] := 4740.03; fTable_C[386, 1] := 6.04791; fTable_C[386, 2] := 0.0301723;
    fTable_C[387, 0] := 4816.69; fTable_C[387, 1] := 6.04667; fTable_C[387, 2] := 0.0291678;
    fTable_C[388, 0] := 4894.60; fTable_C[388, 1] := 6.04547; fTable_C[388, 2] := 0.0281953;
    fTable_C[389, 0] := 4973.77; fTable_C[389, 1] := 6.04429; fTable_C[389, 2] := 0.0272539;
    fTable_C[390, 0] := 5054.21; fTable_C[390, 1] := 6.04313; fTable_C[390, 2] := 0.0263428;
    fTable_C[391, 0] := 5135.96; fTable_C[391, 1] := 6.04200; fTable_C[391, 2] := 0.0254606;
    fTable_C[392, 0] := 5219.03; fTable_C[392, 1] := 6.04090; fTable_C[392, 2] := 0.0246074;
    fTable_C[393, 0] := 5303.44; fTable_C[393, 1] := 6.03983; fTable_C[393, 2] := 0.0237810;
    fTable_C[394, 0] := 5389.22; fTable_C[394, 1] := 6.03877; fTable_C[394, 2] := 0.0229809;
    fTable_C[395, 0] := 5476.39; fTable_C[395, 1] := 6.03774; fTable_C[395, 2] := 0.0222063;
    fTable_C[396, 0] := 5564.97; fTable_C[396, 1] := 6.03674; fTable_C[396, 2] := 0.0214569;
    fTable_C[397, 0] := 5654.98; fTable_C[397, 1] := 6.03576; fTable_C[397, 2] := 0.0207329;
    fTable_C[398, 0] := 5746.44; fTable_C[398, 1] := 6.03480; fTable_C[398, 2] := 0.0200314;
    fTable_C[399, 0] := 5839.39; fTable_C[399, 1] := 6.03386; fTable_C[399, 2] := 0.0193522;
    fTable_C[400, 0] := 5933.83; fTable_C[400, 1] := 6.03295; fTable_C[400, 2] := 0.0186948;
    fTable_C[401, 0] := 6029.81; fTable_C[401, 1] := 6.03205; fTable_C[401, 2] := 0.0180595;
    fTable_C[402, 0] := 6127.33; fTable_C[402, 1] := 6.03118; fTable_C[402, 2] := 0.0174453;
    fTable_C[403, 0] := 6226.44; fTable_C[403, 1] := 6.03033; fTable_C[403, 2] := 0.0168501;
    fTable_C[404, 0] := 6327.15; fTable_C[404, 1] := 6.02950; fTable_C[404, 2] := 0.0162746;
    fTable_C[405, 0] := 6429.48; fTable_C[405, 1] := 6.02869; fTable_C[405, 2] := 0.0157180;
    fTable_C[406, 0] := 6533.48; fTable_C[406, 1] := 6.02789; fTable_C[406, 2] := 0.0151795;
    fTable_C[407, 0] := 6639.15; fTable_C[407, 1] := 6.02712; fTable_C[407, 2] := 0.0146587;
    fTable_C[408, 0] := 6746.54; fTable_C[408, 1] := 6.02637; fTable_C[408, 2] := 0.0141549;
    fTable_C[409, 0] := 6855.65; fTable_C[409, 1] := 6.02563; fTable_C[409, 2] := 0.0136678;
    fTable_C[410, 0] := 6966.54; fTable_C[410, 1] := 6.02491; fTable_C[410, 2] := 0.0131966;
    fTable_C[411, 0] := 7079.22; fTable_C[411, 1] := 6.02421; fTable_C[411, 2] := 0.0127407;
    fTable_C[412, 0] := 7193.72; fTable_C[412, 1] := 6.02352; fTable_C[412, 2] := 0.0123000;
    fTable_C[413, 0] := 7310.07; fTable_C[413, 1] := 6.02285; fTable_C[413, 2] := 0.0118738;
    fTable_C[414, 0] := 7428.31; fTable_C[414, 1] := 6.02220; fTable_C[414, 2] := 0.0114619;
    fTable_C[415, 0] := 7548.45; fTable_C[415, 1] := 6.02156; fTable_C[415, 2] := 0.0110634;
    fTable_C[416, 0] := 7670.54; fTable_C[416, 1] := 6.02094; fTable_C[416, 2] := 0.0106782;
    fTable_C[417, 0] := 7794.61; fTable_C[417, 1] := 6.02034; fTable_C[417, 2] := 0.0103059;
    fTable_C[418, 0] := 7920.68; fTable_C[418, 1] := 6.01975; fTable_C[418, 2] := 0.00994583;
    fTable_C[419, 0] := 8048.79; fTable_C[419, 1] := 6.01917; fTable_C[419, 2] := 0.00959775;
    fTable_C[420, 0] := 8178.98; fTable_C[420, 1] := 6.01861; fTable_C[420, 2] := 0.00926134;
    fTable_C[421, 0] := 8311.26; fTable_C[421, 1] := 6.01806; fTable_C[421, 2] := 0.00893624;
    fTable_C[422, 0] := 8445.69; fTable_C[422, 1] := 6.01753; fTable_C[422, 2] := 0.00862190;
    fTable_C[423, 0] := 8582.29; fTable_C[423, 1] := 6.01700; fTable_C[423, 2] := 0.00831820;
    fTable_C[424, 0] := 8721.11; fTable_C[424, 1] := 6.01650; fTable_C[424, 2] := 0.00802475;
    fTable_C[425, 0] := 8862.16; fTable_C[425, 1] := 6.01600; fTable_C[425, 2] := 0.00774104;
    fTable_C[426, 0] := 9005.50; fTable_C[426, 1] := 6.01552; fTable_C[426, 2] := 0.00746686;
    fTable_C[427, 0] := 9151.16; fTable_C[427, 1] := 6.01505; fTable_C[427, 2] := 0.00720204;
    fTable_C[428, 0] := 9299.17; fTable_C[428, 1] := 6.01459; fTable_C[428, 2] := 0.00694614;
    fTable_C[429, 0] := 9449.58; fTable_C[429, 1] := 6.01414; fTable_C[429, 2] := 0.00669902;
    fTable_C[430, 0] := 9602.42; fTable_C[430, 1] := 6.01370; fTable_C[430, 2] := 0.00646026;
    fTable_C[431, 0] := 9757.73; fTable_C[431, 1] := 6.01328; fTable_C[431, 2] := 0.00622938;
    fTable_C[432, 0] := 9915.55; fTable_C[432, 1] := 6.01286; fTable_C[432, 2] := 0.00600659;
    fTable_C[433, 0] := 10075.9; fTable_C[433, 1] := 6.01246; fTable_C[433, 2] := 0.00579136;
    fTable_C[434, 0] := 10238.9; fTable_C[434, 1] := 6.01206; fTable_C[434, 2] := 0.00558350;
    fTable_C[435, 0] := 10404.5; fTable_C[435, 1] := 6.01168; fTable_C[435, 2] := 0.00538276;
    fTable_C[436, 0] := 10572.8; fTable_C[436, 1] := 6.01131; fTable_C[436, 2] := 0.00518891;
    fTable_C[437, 0] := 10743.8; fTable_C[437, 1] := 6.01094; fTable_C[437, 2] := 0.00500173;
    fTable_C[438, 0] := 10917.6; fTable_C[438, 1] := 6.01059; fTable_C[438, 2] := 0.00482101;
    fTable_C[439, 0] := 11094.2; fTable_C[439, 1] := 6.01024; fTable_C[439, 2] := 0.00464654;
    fTable_C[440, 0] := 11273.6; fTable_C[440, 1] := 6.00991; fTable_C[440, 2] := 0.00447810;
    fTable_C[441, 0] := 11455.9; fTable_C[441, 1] := 6.00958; fTable_C[441, 2] := 0.00431552;
    fTable_C[442, 0] := 11641.2; fTable_C[442, 1] := 6.00926; fTable_C[442, 2] := 0.00415859;
    fTable_C[443, 0] := 11829.5; fTable_C[443, 1] := 6.00895; fTable_C[443, 2] := 0.00400712;
    fTable_C[444, 0] := 12020.8; fTable_C[444, 1] := 6.00864; fTable_C[444, 2] := 0.00386096;
    fTable_C[445, 0] := 12215.3; fTable_C[445, 1] := 6.00835; fTable_C[445, 2] := 0.00371991;
    fTable_C[446, 0] := 12412.8; fTable_C[446, 1] := 6.00806; fTable_C[446, 2] := 0.00358382;
    fTable_C[447, 0] := 12613.6; fTable_C[447, 1] := 6.00778; fTable_C[447, 2] := 0.00345251;
    fTable_C[448, 0] := 12817.6; fTable_C[448, 1] := 6.00751; fTable_C[448, 2] := 0.00332584;
    fTable_C[449, 0] := 13025.0; fTable_C[449, 1] := 6.00724; fTable_C[449, 2] := 0.00320365;
    fTable_C[450, 0] := 13235.6; fTable_C[450, 1] := 6.00698; fTable_C[450, 2] := 0.00308580;
    fTable_C[451, 0] := 13449.7; fTable_C[451, 1] := 6.00673; fTable_C[451, 2] := 0.00297213;
    fTable_C[452, 0] := 13667.2; fTable_C[452, 1] := 6.00648; fTable_C[452, 2] := 0.00286252;
    fTable_C[453, 0] := 13888.3; fTable_C[453, 1] := 6.00625; fTable_C[453, 2] := 0.00275683;
    fTable_C[454, 0] := 14112.9; fTable_C[454, 1] := 6.00601; fTable_C[454, 2] := 0.00265492;
    fTable_C[455, 0] := 14341.2; fTable_C[455, 1] := 6.00579; fTable_C[455, 2] := 0.00255668;
    fTable_C[456, 0] := 14573.1; fTable_C[456, 1] := 6.00557; fTable_C[456, 2] := 0.00246198;
    fTable_C[457, 0] := 14808.9; fTable_C[457, 1] := 6.00535; fTable_C[457, 2] := 0.00237071;
    fTable_C[458, 0] := 15048.4; fTable_C[458, 1] := 6.00514; fTable_C[458, 2] := 0.00228275;
    fTable_C[459, 0] := 15291.8; fTable_C[459, 1] := 6.00494; fTable_C[459, 2] := 0.00219799;
    fTable_C[460, 0] := 15539.1; fTable_C[460, 1] := 6.00474; fTable_C[460, 2] := 0.00211632;
    fTable_C[461, 0] := 15790.4; fTable_C[461, 1] := 6.00455; fTable_C[461, 2] := 0.00203764;
    fTable_C[462, 0] := 16045.8; fTable_C[462, 1] := 6.00436; fTable_C[462, 2] := 0.00196186;
    fTable_C[463, 0] := 16305.4; fTable_C[463, 1] := 6.00418; fTable_C[463, 2] := 0.00188887;
    fTable_C[464, 0] := 16569.1; fTable_C[464, 1] := 6.00400; fTable_C[464, 2] := 0.00181858;
    fTable_C[465, 0] := 16837.1; fTable_C[465, 1] := 6.00383; fTable_C[465, 2] := 0.00175089;
    fTable_C[466, 0] := 17109.4; fTable_C[466, 1] := 6.00366; fTable_C[466, 2] := 0.00168574;
    fTable_C[467, 0] := 17386.1; fTable_C[467, 1] := 6.00350; fTable_C[467, 2] := 0.00162301;
    fTable_C[468, 0] := 17667.4; fTable_C[468, 1] := 6.00334; fTable_C[468, 2] := 0.00156265;
    fTable_C[469, 0] := 17953.1; fTable_C[469, 1] := 6.00319; fTable_C[469, 2] := 0.00150455;
    fTable_C[470, 0] := 18243.5; fTable_C[470, 1] := 6.00304; fTable_C[470, 2] := 0.00144866;
    fTable_C[471, 0] := 18538.6; fTable_C[471, 1] := 6.00289; fTable_C[471, 2] := 0.00139489;
    fTable_C[472, 0] := 18838.4; fTable_C[472, 1] := 6.00275; fTable_C[472, 2] := 0.00134317;
    fTable_C[473, 0] := 19143.1; fTable_C[473, 1] := 6.00261; fTable_C[473, 2] := 0.00129343;
    fTable_C[474, 0] := 19452.7; fTable_C[474, 1] := 6.00248; fTable_C[474, 2] := 0.00124561;
    fTable_C[475, 0] := 19767.4; fTable_C[475, 1] := 6.00235; fTable_C[475, 2] := 0.00119964;
    fTable_C[476, 0] := 20087.1; fTable_C[476, 1] := 6.00222; fTable_C[476, 2] := 0.00116295;
    fTable_C[477, 0] := 20412.0; fTable_C[477, 1] := 6.00211; fTable_C[477, 2] := 0.00111818;
    fTable_C[478, 0] := 20742.1; fTable_C[478, 1] := 6.00199; fTable_C[478, 2] := 0.00107519;
    fTable_C[479, 0] := 21077.6; fTable_C[479, 1] := 6.00187; fTable_C[479, 2] := 0.00103391;
    fTable_C[480, 0] := 21418.5; fTable_C[480, 1] := 6.00176; fTable_C[480, 2] := 0.000994268;
    fTable_C[481, 0] := 21765.0; fTable_C[481, 1] := 6.00165; fTable_C[481, 2] := 0.000956195;
    fTable_C[482, 0] := 22117.0; fTable_C[482, 1] := 6.00154; fTable_C[482, 2] := 0.000919629;
    fTable_C[483, 0] := 22474.7; fTable_C[483, 1] := 6.00144; fTable_C[483, 2] := 0.000884508;
    fTable_C[484, 0] := 22838.2; fTable_C[484, 1] := 6.00134; fTable_C[484, 2] := 0.000850771;
    fTable_C[485, 0] := 23207.6; fTable_C[485, 1] := 6.00124; fTable_C[485, 2] := 0.000818364;
    fTable_C[486, 0] := 23583.0; fTable_C[486, 1] := 6.00115; fTable_C[486, 2] := 0.000787230;
    fTable_C[487, 0] := 23964.4; fTable_C[487, 1] := 6.00105; fTable_C[487, 2] := 0.000757320;
    fTable_C[488, 0] := 24352.0; fTable_C[488, 1] := 6.00096; fTable_C[488, 2] := 0.000728582;
    fTable_C[489, 0] := 24745.9; fTable_C[489, 1] := 6.00088; fTable_C[489, 2] := 0.000700971;
    fTable_C[490, 0] := 25146.2; fTable_C[490, 1] := 6.00079; fTable_C[490, 2] := 0.000674438;
    fTable_C[491, 0] := 25552.9; fTable_C[491, 1] := 6.00071; fTable_C[491, 2] := 0.000648942;
    fTable_C[492, 0] := 25966.2; fTable_C[492, 1] := 6.00063; fTable_C[492, 2] := 0.000624439;
    fTable_C[493, 0] := 26386.1; fTable_C[493, 1] := 6.00055; fTable_C[493, 2] := 0.000600890;
    fTable_C[494, 0] := 26812.9; fTable_C[494, 1] := 6.00048; fTable_C[494, 2] := 0.000578257;
    fTable_C[495, 0] := 27246.6; fTable_C[495, 1] := 6.00040; fTable_C[495, 2] := 0.000556501;
    fTable_C[496, 0] := 27687.3; fTable_C[496, 1] := 6.00033; fTable_C[496, 2] := 0.000535590;
    fTable_C[497, 0] := 28135.1; fTable_C[497, 1] := 6.00026; fTable_C[497, 2] := 0.000515487;
    fTable_C[498, 0] := 28590.2; fTable_C[498, 1] := 6.00020; fTable_C[498, 2] := 0.000496161;
    fTable_C[499, 0] := 29052.6; fTable_C[499, 1] := 6.00013; fTable_C[499, 2] := 0.000477581;
    fTable_C[500, 0] := 29522.5; fTable_C[500, 1] := 6.00007; fTable_C[500, 2] := 0.000459716;
    fTable_C[501, 0] := 30000.0; fTable_C[501, 1] := 6.00000; fTable_C[501, 2] := 0.000442540;

    (* Table initialization: fTable_Al *)
    fTable_Al[0, 0] := 10.0000; fTable_Al[0, 1] := -9999; fTable_Al[0, 2] := 3.11990;
    fTable_Al[1, 0] := 10.1617; fTable_Al[1, 1] := -9999; fTable_Al[1, 2] := 3.05822;
    fTable_Al[2, 0] := 10.3261; fTable_Al[2, 1] := -9999; fTable_Al[2, 2] := 2.99776;
    fTable_Al[3, 0] := 10.4931; fTable_Al[3, 1] := -9999; fTable_Al[3, 2] := 2.93850;
    fTable_Al[4, 0] := 10.6628; fTable_Al[4, 1] := -9999; fTable_Al[4, 2] := 2.88041;
    fTable_Al[5, 0] := 10.8353; fTable_Al[5, 1] := -9999; fTable_Al[5, 2] := 2.82347;
    fTable_Al[6, 0] := 11.0106; fTable_Al[6, 1] := -9999; fTable_Al[6, 2] := 2.76766;
    fTable_Al[7, 0] := 11.1886; fTable_Al[7, 1] := -9999; fTable_Al[7, 2] := 2.72200;
    fTable_Al[8, 0] := 11.3696; fTable_Al[8, 1] := -9999; fTable_Al[8, 2] := 2.69148;
    fTable_Al[9, 0] := 11.5535; fTable_Al[9, 1] := -9999; fTable_Al[9, 2] := 2.66129;
    fTable_Al[10, 0] := 11.7404; fTable_Al[10, 1] := -9999; fTable_Al[10, 2] := 2.63145;
    fTable_Al[11, 0] := 11.9303; fTable_Al[11, 1] := -9999; fTable_Al[11, 2] := 2.60195;
    fTable_Al[12, 0] := 12.1232; fTable_Al[12, 1] := -9999; fTable_Al[12, 2] := 2.57277;
    fTable_Al[13, 0] := 12.3193; fTable_Al[13, 1] := -9999; fTable_Al[13, 2] := 2.54392;
    fTable_Al[14, 0] := 12.5186; fTable_Al[14, 1] := -9999; fTable_Al[14, 2] := 2.51539;
    fTable_Al[15, 0] := 12.7210; fTable_Al[15, 1] := -9999; fTable_Al[15, 2] := 2.46668;
    fTable_Al[16, 0] := 12.9268; fTable_Al[16, 1] := -9999; fTable_Al[16, 2] := 2.41373;
    fTable_Al[17, 0] := 13.1359; fTable_Al[17, 1] := -9999; fTable_Al[17, 2] := 2.36192;
    fTable_Al[18, 0] := 13.3483; fTable_Al[18, 1] := -9999; fTable_Al[18, 2] := 2.30898;
    fTable_Al[19, 0] := 13.5642; fTable_Al[19, 1] := -9999; fTable_Al[19, 2] := 2.23405;
    fTable_Al[20, 0] := 13.7836; fTable_Al[20, 1] := -9999; fTable_Al[20, 2] := 2.15356;
    fTable_Al[21, 0] := 14.0066; fTable_Al[21, 1] := -9999; fTable_Al[21, 2] := 2.06069;
    fTable_Al[22, 0] := 14.2331; fTable_Al[22, 1] := -9999; fTable_Al[22, 2] := 1.96756;
    fTable_Al[23, 0] := 14.4633; fTable_Al[23, 1] := -9999; fTable_Al[23, 2] := 1.81305;
    fTable_Al[24, 0] := 14.6973; fTable_Al[24, 1] := -9999; fTable_Al[24, 2] := 1.35947;
    fTable_Al[25, 0] := 14.9350; fTable_Al[25, 1] := -9999; fTable_Al[25, 2] := 0.902011;
    fTable_Al[26, 0] := 15.1765; fTable_Al[26, 1] := -9999; fTable_Al[26, 2] := 0.609172;
    fTable_Al[27, 0] := 15.4220; fTable_Al[27, 1] := -9999; fTable_Al[27, 2] := 0.439681;
    fTable_Al[28, 0] := 15.6714; fTable_Al[28, 1] := -9999; fTable_Al[28, 2] := 0.372037;
    fTable_Al[29, 0] := 15.9249; fTable_Al[29, 1] := -9999; fTable_Al[29, 2] := 0.326005;
    fTable_Al[30, 0] := 16.1825; fTable_Al[30, 1] := -9999; fTable_Al[30, 2] := 0.285669;
    fTable_Al[31, 0] := 16.4442; fTable_Al[31, 1] := -9999; fTable_Al[31, 2] := 0.247205;
    fTable_Al[32, 0] := 16.7102; fTable_Al[32, 1] := -9999; fTable_Al[32, 2] := 0.213520;
    fTable_Al[33, 0] := 16.9805; fTable_Al[33, 1] := -9999; fTable_Al[33, 2] := 0.196522;
    fTable_Al[34, 0] := 17.2551; fTable_Al[34, 1] := -9999; fTable_Al[34, 2] := 0.181095;
    fTable_Al[35, 0] := 17.5342; fTable_Al[35, 1] := -9999; fTable_Al[35, 2] := 0.168385;
    fTable_Al[36, 0] := 17.8178; fTable_Al[36, 1] := -9999; fTable_Al[36, 2] := 0.160808;
    fTable_Al[37, 0] := 18.1060; fTable_Al[37, 1] := -9999; fTable_Al[37, 2] := 0.153573;
    fTable_Al[38, 0] := 18.3989; fTable_Al[38, 1] := -9999; fTable_Al[38, 2] := 0.146663;
    fTable_Al[39, 0] := 18.6964; fTable_Al[39, 1] := -9999; fTable_Al[39, 2] := 0.140063;
    fTable_Al[40, 0] := 18.9988; fTable_Al[40, 1] := -9999; fTable_Al[40, 2] := 0.133164;
    fTable_Al[41, 0] := 19.3061; fTable_Al[41, 1] := -9999; fTable_Al[41, 2] := 0.126575;
    fTable_Al[42, 0] := 19.6184; fTable_Al[42, 1] := -9999; fTable_Al[42, 2] := 0.120312;
    fTable_Al[43, 0] := 19.9357; fTable_Al[43, 1] := -9999; fTable_Al[43, 2] := 0.114360;
    fTable_Al[44, 0] := 20.2582; fTable_Al[44, 1] := -9999; fTable_Al[44, 2] := 0.109752;
    fTable_Al[45, 0] := 20.5858; fTable_Al[45, 1] := -9999; fTable_Al[45, 2] := 0.111010;
    fTable_Al[46, 0] := 20.9188; fTable_Al[46, 1] := -9999; fTable_Al[46, 2] := 0.112282;
    fTable_Al[47, 0] := 21.2571; fTable_Al[47, 1] := -9999; fTable_Al[47, 2] := 0.113569;
    fTable_Al[48, 0] := 21.6009; fTable_Al[48, 1] := -9999; fTable_Al[48, 2] := 0.114870;
    fTable_Al[49, 0] := 21.9503; fTable_Al[49, 1] := -9999; fTable_Al[49, 2] := 0.116186;
    fTable_Al[50, 0] := 22.3053; fTable_Al[50, 1] := -9999; fTable_Al[50, 2] := 0.117518;
    fTable_Al[51, 0] := 22.6661; fTable_Al[51, 1] := -9999; fTable_Al[51, 2] := 0.118864;
    fTable_Al[52, 0] := 23.0327; fTable_Al[52, 1] := -9999; fTable_Al[52, 2] := 0.120227;
    fTable_Al[53, 0] := 23.4053; fTable_Al[53, 1] := -9999; fTable_Al[53, 2] := 0.122751;
    fTable_Al[54, 0] := 23.7838; fTable_Al[54, 1] := -9999; fTable_Al[54, 2] := 0.126315;
    fTable_Al[55, 0] := 24.1685; fTable_Al[55, 1] := -9999; fTable_Al[55, 2] := 0.129984;
    fTable_Al[56, 0] := 24.5594; fTable_Al[56, 1] := -9999; fTable_Al[56, 2] := 0.133759;
    fTable_Al[57, 0] := 24.9566; fTable_Al[57, 1] := -9999; fTable_Al[57, 2] := 0.137643;
    fTable_Al[58, 0] := 25.3603; fTable_Al[58, 1] := -9999; fTable_Al[58, 2] := 0.141640;
    fTable_Al[59, 0] := 25.7705; fTable_Al[59, 1] := -9999; fTable_Al[59, 2] := 0.145495;
    fTable_Al[60, 0] := 26.1873; fTable_Al[60, 1] := -9999; fTable_Al[60, 2] := 0.148244;
    fTable_Al[61, 0] := 26.6109; fTable_Al[61, 1] := -9999; fTable_Al[61, 2] := 0.151045;
    fTable_Al[62, 0] := 27.0413; fTable_Al[62, 1] := -9999; fTable_Al[62, 2] := 0.153898;
    fTable_Al[63, 0] := 27.4786; fTable_Al[63, 1] := -9999; fTable_Al[63, 2] := 0.156806;
    fTable_Al[64, 0] := 27.9231; fTable_Al[64, 1] := -9999; fTable_Al[64, 2] := 0.159768;
    fTable_Al[65, 0] := 28.3747; fTable_Al[65, 1] := -9999; fTable_Al[65, 2] := 0.162787;
    fTable_Al[66, 0] := 28.8337; fTable_Al[66, 1] := -9999; fTable_Al[66, 2] := 0.165863;
    fTable_Al[67, 0] := 29.3000; fTable_Al[67, 1] := 2.34285; fTable_Al[67, 2] := 0.168996;
    fTable_Al[68, 0] := 29.7739; fTable_Al[68, 1] := 2.32717; fTable_Al[68, 2] := 0.172189;
    fTable_Al[69, 0] := 30.2555; fTable_Al[69, 1] := 2.31139; fTable_Al[69, 2] := 0.175442;
    fTable_Al[70, 0] := 30.7449; fTable_Al[70, 1] := 2.29552; fTable_Al[70, 2] := 0.178757;
    fTable_Al[71, 0] := 31.2421; fTable_Al[71, 1] := 2.27956; fTable_Al[71, 2] := 0.182134;
    fTable_Al[72, 0] := 31.7475; fTable_Al[72, 1] := 2.26350; fTable_Al[72, 2] := 0.185575;
    fTable_Al[73, 0] := 32.2609; fTable_Al[73, 1] := 2.24754; fTable_Al[73, 2] := 0.189081;
    fTable_Al[74, 0] := 32.7827; fTable_Al[74, 1] := 2.23175; fTable_Al[74, 2] := 0.192378;
    fTable_Al[75, 0] := 33.3130; fTable_Al[75, 1] := 2.21555; fTable_Al[75, 2] := 0.194561;
    fTable_Al[76, 0] := 33.8518; fTable_Al[76, 1] := 2.19843; fTable_Al[76, 2] := 0.196767;
    fTable_Al[77, 0] := 34.3993; fTable_Al[77, 1] := 2.18068; fTable_Al[77, 2] := 0.198999;
    fTable_Al[78, 0] := 34.9557; fTable_Al[78, 1] := 2.16235; fTable_Al[78, 2] := 0.201256;
    fTable_Al[79, 0] := 35.5211; fTable_Al[79, 1] := 2.14342; fTable_Al[79, 2] := 0.203539;
    fTable_Al[80, 0] := 36.0956; fTable_Al[80, 1] := 2.12388; fTable_Al[80, 2] := 0.205847;
    fTable_Al[81, 0] := 36.6794; fTable_Al[81, 1] := 2.10371; fTable_Al[81, 2] := 0.208182;
    fTable_Al[82, 0] := 37.2727; fTable_Al[82, 1] := 2.08287; fTable_Al[82, 2] := 0.210544;
    fTable_Al[83, 0] := 37.8755; fTable_Al[83, 1] := 2.06135; fTable_Al[83, 2] := 0.212932;
    fTable_Al[84, 0] := 38.4882; fTable_Al[84, 1] := 2.03911; fTable_Al[84, 2] := 0.215347;
    fTable_Al[85, 0] := 39.1107; fTable_Al[85, 1] := 2.01612; fTable_Al[85, 2] := 0.217789;
    fTable_Al[86, 0] := 39.7432; fTable_Al[86, 1] := 1.99237; fTable_Al[86, 2] := 0.220259;
    fTable_Al[87, 0] := 40.3861; fTable_Al[87, 1] := 1.96797; fTable_Al[87, 2] := 0.222758;
    fTable_Al[88, 0] := 41.0393; fTable_Al[88, 1] := 1.94295; fTable_Al[88, 2] := 0.225068;
    fTable_Al[89, 0] := 41.7031; fTable_Al[89, 1] := 1.91682; fTable_Al[89, 2] := 0.226470;
    fTable_Al[90, 0] := 42.3776; fTable_Al[90, 1] := 1.88912; fTable_Al[90, 2] := 0.227880;
    fTable_Al[91, 0] := 43.0630; fTable_Al[91, 1] := 1.86007; fTable_Al[91, 2] := 0.229299;
    fTable_Al[92, 0] := 43.7595; fTable_Al[92, 1] := 1.82966; fTable_Al[92, 2] := 0.230727;
    fTable_Al[93, 0] := 44.4673; fTable_Al[93, 1] := 1.79787; fTable_Al[93, 2] := 0.232164;
    fTable_Al[94, 0] := 45.1865; fTable_Al[94, 1] := 1.76466; fTable_Al[94, 2] := 0.233610;
    fTable_Al[95, 0] := 45.9174; fTable_Al[95, 1] := 1.73005; fTable_Al[95, 2] := 0.235064;
    fTable_Al[96, 0] := 46.6600; fTable_Al[96, 1] := 1.69399; fTable_Al[96, 2] := 0.236528;
    fTable_Al[97, 0] := 47.4147; fTable_Al[97, 1] := 1.65814; fTable_Al[97, 2] := 0.238001;
    fTable_Al[98, 0] := 48.1816; fTable_Al[98, 1] := 1.62074; fTable_Al[98, 2] := 0.235842;
    fTable_Al[99, 0] := 48.9609; fTable_Al[99, 1] := 1.57843; fTable_Al[99, 2] := 0.232104;
    fTable_Al[100, 0] := 49.7528; fTable_Al[100, 1] := 1.53229; fTable_Al[100, 2] := 0.228425;
    fTable_Al[101, 0] := 50.5576; fTable_Al[101, 1] := 1.48252; fTable_Al[101, 2] := 0.224805;
    fTable_Al[102, 0] := 51.3753; fTable_Al[102, 1] := 1.42904; fTable_Al[102, 2] := 0.221242;
    fTable_Al[103, 0] := 52.2062; fTable_Al[103, 1] := 1.37159; fTable_Al[103, 2] := 0.217735;
    fTable_Al[104, 0] := 53.0506; fTable_Al[104, 1] := 1.30972; fTable_Al[104, 2] := 0.214284;
    fTable_Al[105, 0] := 53.9087; fTable_Al[105, 1] := 1.24315; fTable_Al[105, 2] := 0.211759;
    fTable_Al[106, 0] := 54.7806; fTable_Al[106, 1] := 1.17229; fTable_Al[106, 2] := 0.209829;
    fTable_Al[107, 0] := 55.6667; fTable_Al[107, 1] := 1.09675; fTable_Al[107, 2] := 0.207917;
    fTable_Al[108, 0] := 56.5670; fTable_Al[108, 1] := 1.01559; fTable_Al[108, 2] := 0.206022;
    fTable_Al[109, 0] := 57.4820; fTable_Al[109, 1] := 0.928103; fTable_Al[109, 2] := 0.204145;
    fTable_Al[110, 0] := 58.4117; fTable_Al[110, 1] := 0.833427; fTable_Al[110, 2] := 0.202284;
    fTable_Al[111, 0] := 59.3564; fTable_Al[111, 1] := 0.729805; fTable_Al[111, 2] := 0.200441;
    fTable_Al[112, 0] := 60.3165; fTable_Al[112, 1] := 0.616720; fTable_Al[112, 2] := 0.200207;
    fTable_Al[113, 0] := 61.2921; fTable_Al[113, 1] := 0.494009; fTable_Al[113, 2] := 0.200602;
    fTable_Al[114, 0] := 62.2834; fTable_Al[114, 1] := 0.359171; fTable_Al[114, 2] := 0.200998;
    fTable_Al[115, 0] := 63.2908; fTable_Al[115, 1] := 0.206766; fTable_Al[115, 2] := 0.201394;
    fTable_Al[116, 0] := 64.3145; fTable_Al[116, 1] := 0.0367838; fTable_Al[116, 2] := 0.208215;
    fTable_Al[117, 0] := 65.3547; fTable_Al[117, 1] := -0.150100; fTable_Al[117, 2] := 0.215821;
    fTable_Al[118, 0] := 66.4118; fTable_Al[118, 1] := -0.363400; fTable_Al[118, 2] := 0.223705;
    fTable_Al[119, 0] := 67.4859; fTable_Al[119, 1] := -0.612251; fTable_Al[119, 2] := 0.231878;
    fTable_Al[120, 0] := 68.5775; fTable_Al[120, 1] := -0.913185; fTable_Al[120, 2] := 0.239512;
    fTable_Al[121, 0] := 69.6867; fTable_Al[121, 1] := -1.29772; fTable_Al[121, 2] := 0.247287;
    fTable_Al[122, 0] := 70.8138; fTable_Al[122, 1] := -1.83916; fTable_Al[122, 2] := 0.255315;
    fTable_Al[123, 0] := 71.9591; fTable_Al[123, 1] := -2.82640; fTable_Al[123, 2] := 0.263603;
    fTable_Al[124, 0] := 72.6000; fTable_Al[124, 1] := -4.71870; fTable_Al[124, 2] := 0.268298;
    fTable_Al[125, 0] := 72.8000; fTable_Al[125, 1] := -4.77865; fTable_Al[125, 2] := 3.05391;
    fTable_Al[126, 0] := 73.1230; fTable_Al[126, 1] := -3.57738; fTable_Al[126, 2] := 3.10106;
    fTable_Al[127, 0] := 74.3057; fTable_Al[127, 1] := -2.58986; fTable_Al[127, 2] := 3.27808;
    fTable_Al[128, 0] := 75.5076; fTable_Al[128, 1] := -2.24498; fTable_Al[128, 2] := 3.46521;
    fTable_Al[129, 0] := 76.7289; fTable_Al[129, 1] := -2.04974; fTable_Al[129, 2] := 3.66301;
    fTable_Al[130, 0] := 77.9699; fTable_Al[130, 1] := -1.91658; fTable_Al[130, 2] := 3.87212;
    fTable_Al[131, 0] := 79.2310; fTable_Al[131, 1] := -1.81173; fTable_Al[131, 2] := 4.09316;
    fTable_Al[132, 0] := 80.5125; fTable_Al[132, 1] := -1.71207; fTable_Al[132, 2] := 4.32681;
    fTable_Al[133, 0] := 81.8147; fTable_Al[133, 1] := -1.61278; fTable_Al[133, 2] := 4.55877;
    fTable_Al[134, 0] := 83.1380; fTable_Al[134, 1] := -1.51695; fTable_Al[134, 2] := 4.80227;
    fTable_Al[135, 0] := 84.4827; fTable_Al[135, 1] := -1.40821; fTable_Al[135, 2] := 5.05877;
    fTable_Al[136, 0] := 85.8491; fTable_Al[136, 1] := -1.24639; fTable_Al[136, 2] := 5.32897;
    fTable_Al[137, 0] := 87.2377; fTable_Al[137, 1] := -1.04412; fTable_Al[137, 2] := 5.54566;
    fTable_Al[138, 0] := 88.6487; fTable_Al[138, 1] := -0.869623; fTable_Al[138, 2] := 5.69070;
    fTable_Al[139, 0] := 90.0825; fTable_Al[139, 1] := -0.729715; fTable_Al[139, 2] := 5.83953;
    fTable_Al[140, 0] := 91.5395; fTable_Al[140, 1] := -0.602517; fTable_Al[140, 2] := 5.99225;
    fTable_Al[141, 0] := 93.0201; fTable_Al[141, 1] := -0.481649; fTable_Al[141, 2] := 6.14897;
    fTable_Al[142, 0] := 94.5246; fTable_Al[142, 1] := -0.363849; fTable_Al[142, 2] := 6.30978;
    fTable_Al[143, 0] := 96.0535; fTable_Al[143, 1] := -0.246485; fTable_Al[143, 2] := 6.47480;
    fTable_Al[144, 0] := 97.6071; fTable_Al[144, 1] := -0.127798; fTable_Al[144, 2] := 6.64413;
    fTable_Al[145, 0] := 99.1858; fTable_Al[145, 1] := -0.00572152; fTable_Al[145, 2] := 6.81790;
    fTable_Al[146, 0] := 100.790; fTable_Al[146, 1] := 0.121587; fTable_Al[146, 2] := 6.99620;
    fTable_Al[147, 0] := 102.420; fTable_Al[147, 1] := 0.257648; fTable_Al[147, 2] := 7.17918;
    fTable_Al[148, 0] := 104.077; fTable_Al[148, 1] := 0.408417; fTable_Al[148, 2] := 7.36022;
    fTable_Al[149, 0] := 105.760; fTable_Al[149, 1] := 0.563135; fTable_Al[149, 2] := 7.52866;
    fTable_Al[150, 0] := 107.471; fTable_Al[150, 1] := 0.713525; fTable_Al[150, 2] := 7.70096;
    fTable_Al[151, 0] := 109.209; fTable_Al[151, 1] := 0.869599; fTable_Al[151, 2] := 7.87720;
    fTable_Al[152, 0] := 110.975; fTable_Al[152, 1] := 1.03257; fTable_Al[152, 2] := 8.05748;
    fTable_Al[153, 0] := 112.770; fTable_Al[153, 1] := 1.20465; fTable_Al[153, 2] := 8.24188;
    fTable_Al[154, 0] := 114.594; fTable_Al[154, 1] := 1.38785; fTable_Al[154, 2] := 8.43050;
    fTable_Al[155, 0] := 116.448; fTable_Al[155, 1] := 1.58511; fTable_Al[155, 2] := 8.62344;
    fTable_Al[156, 0] := 118.331; fTable_Al[156, 1] := 1.79993; fTable_Al[156, 2] := 8.82080;
    fTable_Al[157, 0] := 120.245; fTable_Al[157, 1] := 2.03832; fTable_Al[157, 2] := 9.02267;
    fTable_Al[158, 0] := 122.190; fTable_Al[158, 1] := 2.31105; fTable_Al[158, 2] := 9.22916;
    fTable_Al[159, 0] := 124.166; fTable_Al[159, 1] := 2.65726; fTable_Al[159, 2] := 9.44037;
    fTable_Al[160, 0] := 126.175; fTable_Al[160, 1] := 3.05450; fTable_Al[160, 2] := 9.49754;
    fTable_Al[161, 0] := 128.215; fTable_Al[161, 1] := 3.37636; fTable_Al[161, 2] := 9.51114;
    fTable_Al[162, 0] := 130.289; fTable_Al[162, 1] := 3.65455; fTable_Al[162, 2] := 9.52475;
    fTable_Al[163, 0] := 132.397; fTable_Al[163, 1] := 3.91635; fTable_Al[163, 2] := 9.53840;
    fTable_Al[164, 0] := 134.538; fTable_Al[164, 1] := 4.16654; fTable_Al[164, 2] := 9.55206;
    fTable_Al[165, 0] := 136.714; fTable_Al[165, 1] := 4.40886; fTable_Al[165, 2] := 9.56573;
    fTable_Al[166, 0] := 138.925; fTable_Al[166, 1] := 4.64594; fTable_Al[166, 2] := 9.57943;
    fTable_Al[167, 0] := 141.172; fTable_Al[167, 1] := 4.87987; fTable_Al[167, 2] := 9.59315;
    fTable_Al[168, 0] := 143.456; fTable_Al[168, 1] := 5.11258; fTable_Al[168, 2] := 9.60689;
    fTable_Al[169, 0] := 145.776; fTable_Al[169, 1] := 5.34618; fTable_Al[169, 2] := 9.62064;
    fTable_Al[170, 0] := 148.134; fTable_Al[170, 1] := 5.58438; fTable_Al[170, 2] := 9.63443;
    fTable_Al[171, 0] := 150.530; fTable_Al[171, 1] := 5.83549; fTable_Al[171, 2] := 9.64822;
    fTable_Al[172, 0] := 152.964; fTable_Al[172, 1] := 6.09089; fTable_Al[172, 2] := 9.62310;
    fTable_Al[173, 0] := 155.439; fTable_Al[173, 1] := 6.32655; fTable_Al[173, 2] := 9.59689;
    fTable_Al[174, 0] := 157.953; fTable_Al[174, 1] := 6.55613; fTable_Al[174, 2] := 9.57075;
    fTable_Al[175, 0] := 160.507; fTable_Al[175, 1] := 6.78302; fTable_Al[175, 2] := 9.54468;
    fTable_Al[176, 0] := 163.103; fTable_Al[176, 1] := 7.00948; fTable_Al[176, 2] := 9.51868;
    fTable_Al[177, 0] := 165.742; fTable_Al[177, 1] := 7.23759; fTable_Al[177, 2] := 9.49275;
    fTable_Al[178, 0] := 168.422; fTable_Al[178, 1] := 7.46980; fTable_Al[178, 2] := 9.46689;
    fTable_Al[179, 0] := 171.146; fTable_Al[179, 1] := 7.70942; fTable_Al[179, 2] := 9.44111;
    fTable_Al[180, 0] := 173.915; fTable_Al[180, 1] := 7.96219; fTable_Al[180, 2] := 9.41540;
    fTable_Al[181, 0] := 176.727; fTable_Al[181, 1] := 8.24313; fTable_Al[181, 2] := 9.38975;
    fTable_Al[182, 0] := 179.586; fTable_Al[182, 1] := 8.57964; fTable_Al[182, 2] := 9.31472;
    fTable_Al[183, 0] := 182.491; fTable_Al[183, 1] := 8.88946; fTable_Al[183, 2] := 9.13115;
    fTable_Al[184, 0] := 185.442; fTable_Al[184, 1] := 9.11623; fTable_Al[184, 2] := 8.95119;
    fTable_Al[185, 0] := 188.442; fTable_Al[185, 1] := 9.32069; fTable_Al[185, 2] := 8.77477;
    fTable_Al[186, 0] := 191.489; fTable_Al[186, 1] := 9.50496; fTable_Al[186, 2] := 8.60184;
    fTable_Al[187, 0] := 194.587; fTable_Al[187, 1] := 9.67311; fTable_Al[187, 2] := 8.43231;
    fTable_Al[188, 0] := 197.734; fTable_Al[188, 1] := 9.82798; fTable_Al[188, 2] := 8.26612;
    fTable_Al[189, 0] := 200.932; fTable_Al[189, 1] := 9.97197; fTable_Al[189, 2] := 8.10317;
    fTable_Al[190, 0] := 204.182; fTable_Al[190, 1] := 10.1053; fTable_Al[190, 2] := 7.93953;
    fTable_Al[191, 0] := 207.485; fTable_Al[191, 1] := 10.2265; fTable_Al[191, 2] := 7.77920;
    fTable_Al[192, 0] := 210.840; fTable_Al[192, 1] := 10.3376; fTable_Al[192, 2] := 7.62210;
    fTable_Al[193, 0] := 214.251; fTable_Al[193, 1] := 10.4388; fTable_Al[193, 2] := 7.46817;
    fTable_Al[194, 0] := 217.716; fTable_Al[194, 1] := 10.5299; fTable_Al[194, 2] := 7.31736;
    fTable_Al[195, 0] := 221.237; fTable_Al[195, 1] := 10.6083; fTable_Al[195, 2] := 7.16959;
    fTable_Al[196, 0] := 224.816; fTable_Al[196, 1] := 10.6680; fTable_Al[196, 2] := 7.03532;
    fTable_Al[197, 0] := 228.452; fTable_Al[197, 1] := 10.7284; fTable_Al[197, 2] := 6.92993;
    fTable_Al[198, 0] := 232.147; fTable_Al[198, 1] := 10.8042; fTable_Al[198, 2] := 6.82611;
    fTable_Al[199, 0] := 235.902; fTable_Al[199, 1] := 10.8811; fTable_Al[199, 2] := 6.72384;
    fTable_Al[200, 0] := 239.717; fTable_Al[200, 1] := 10.9592; fTable_Al[200, 2] := 6.62312;
    fTable_Al[201, 0] := 243.595; fTable_Al[201, 1] := 11.0380; fTable_Al[201, 2] := 6.52389;
    fTable_Al[202, 0] := 247.535; fTable_Al[202, 1] := 11.1176; fTable_Al[202, 2] := 6.42616;
    fTable_Al[203, 0] := 251.538; fTable_Al[203, 1] := 11.1983; fTable_Al[203, 2] := 6.32988;
    fTable_Al[204, 0] := 255.607; fTable_Al[204, 1] := 11.2808; fTable_Al[204, 2] := 6.23505;
    fTable_Al[205, 0] := 259.741; fTable_Al[205, 1] := 11.3664; fTable_Al[205, 2] := 6.14164;
    fTable_Al[206, 0] := 263.942; fTable_Al[206, 1] := 11.4630; fTable_Al[206, 2] := 6.04964;
    fTable_Al[207, 0] := 268.211; fTable_Al[207, 1] := 11.5725; fTable_Al[207, 2] := 5.94856;
    fTable_Al[208, 0] := 272.549; fTable_Al[208, 1] := 11.6747; fTable_Al[208, 2] := 5.80523;
    fTable_Al[209, 0] := 276.957; fTable_Al[209, 1] := 11.7511; fTable_Al[209, 2] := 5.66535;
    fTable_Al[210, 0] := 281.437; fTable_Al[210, 1] := 11.8159; fTable_Al[210, 2] := 5.52884;
    fTable_Al[211, 0] := 285.989; fTable_Al[211, 1] := 11.8724; fTable_Al[211, 2] := 5.39563;
    fTable_Al[212, 0] := 290.615; fTable_Al[212, 1] := 11.9222; fTable_Al[212, 2] := 5.26561;
    fTable_Al[213, 0] := 295.315; fTable_Al[213, 1] := 11.9664; fTable_Al[213, 2] := 5.13874;
    fTable_Al[214, 0] := 300.092; fTable_Al[214, 1] := 12.0058; fTable_Al[214, 2] := 5.01492;
    fTable_Al[215, 0] := 304.945; fTable_Al[215, 1] := 12.0408; fTable_Al[215, 2] := 4.89409;
    fTable_Al[216, 0] := 309.878; fTable_Al[216, 1] := 12.0718; fTable_Al[216, 2] := 4.77616;
    fTable_Al[217, 0] := 314.890; fTable_Al[217, 1] := 12.0993; fTable_Al[217, 2] := 4.66108;
    fTable_Al[218, 0] := 319.983; fTable_Al[218, 1] := 12.1235; fTable_Al[218, 2] := 4.54877;
    fTable_Al[219, 0] := 325.158; fTable_Al[219, 1] := 12.1445; fTable_Al[219, 2] := 4.43917;
    fTable_Al[220, 0] := 330.418; fTable_Al[220, 1] := 12.1625; fTable_Al[220, 2] := 4.33221;
    fTable_Al[221, 0] := 335.762; fTable_Al[221, 1] := 12.1777; fTable_Al[221, 2] := 4.22782;
    fTable_Al[222, 0] := 341.192; fTable_Al[222, 1] := 12.1900; fTable_Al[222, 2] := 4.12595;
    fTable_Al[223, 0] := 346.711; fTable_Al[223, 1] := 12.1992; fTable_Al[223, 2] := 4.02654;
    fTable_Al[224, 0] := 352.319; fTable_Al[224, 1] := 12.2049; fTable_Al[224, 2] := 3.92952;
    fTable_Al[225, 0] := 358.017; fTable_Al[225, 1] := 12.2045; fTable_Al[225, 2] := 3.83484;
    fTable_Al[226, 0] := 363.808; fTable_Al[226, 1] := 12.1998; fTable_Al[226, 2] := 3.75388;
    fTable_Al[227, 0] := 369.692; fTable_Al[227, 1] := 12.2008; fTable_Al[227, 2] := 3.67818;
    fTable_Al[228, 0] := 375.672; fTable_Al[228, 1] := 12.2048; fTable_Al[228, 2] := 3.60400;
    fTable_Al[229, 0] := 381.748; fTable_Al[229, 1] := 12.2097; fTable_Al[229, 2] := 3.53133;
    fTable_Al[230, 0] := 387.922; fTable_Al[230, 1] := 12.2152; fTable_Al[230, 2] := 3.46011;
    fTable_Al[231, 0] := 394.197; fTable_Al[231, 1] := 12.2210; fTable_Al[231, 2] := 3.39034;
    fTable_Al[232, 0] := 400.573; fTable_Al[232, 1] := 12.2270; fTable_Al[232, 2] := 3.32197;
    fTable_Al[233, 0] := 407.052; fTable_Al[233, 1] := 12.2333; fTable_Al[233, 2] := 3.25498;
    fTable_Al[234, 0] := 413.635; fTable_Al[234, 1] := 12.2399; fTable_Al[234, 2] := 3.18934;
    fTable_Al[235, 0] := 420.326; fTable_Al[235, 1] := 12.2470; fTable_Al[235, 2] := 3.12502;
    fTable_Al[236, 0] := 427.124; fTable_Al[236, 1] := 12.2549; fTable_Al[236, 2] := 3.06201;
    fTable_Al[237, 0] := 434.032; fTable_Al[237, 1] := 12.2652; fTable_Al[237, 2] := 3.00026;
    fTable_Al[238, 0] := 441.052; fTable_Al[238, 1] := 12.2773; fTable_Al[238, 2] := 2.93296;
    fTable_Al[239, 0] := 448.186; fTable_Al[239, 1] := 12.2849; fTable_Al[239, 2] := 2.86424;
    fTable_Al[240, 0] := 455.435; fTable_Al[240, 1] := 12.2892; fTable_Al[240, 2] := 2.79730;
    fTable_Al[241, 0] := 462.802; fTable_Al[241, 1] := 12.2920; fTable_Al[241, 2] := 2.73189;
    fTable_Al[242, 0] := 470.287; fTable_Al[242, 1] := 12.2937; fTable_Al[242, 2] := 2.66798;
    fTable_Al[243, 0] := 477.894; fTable_Al[243, 1] := 12.2943; fTable_Al[243, 2] := 2.60559;
    fTable_Al[244, 0] := 485.623; fTable_Al[244, 1] := 12.2945; fTable_Al[244, 2] := 2.54463;
    fTable_Al[245, 0] := 493.478; fTable_Al[245, 1] := 12.2942; fTable_Al[245, 2] := 2.48490;
    fTable_Al[246, 0] := 501.459; fTable_Al[246, 1] := 12.2939; fTable_Al[246, 2] := 2.42570;
    fTable_Al[247, 0] := 509.570; fTable_Al[247, 1] := 12.2928; fTable_Al[247, 2] := 2.36643;
    fTable_Al[248, 0] := 517.812; fTable_Al[248, 1] := 12.2896; fTable_Al[248, 2] := 2.30801;
    fTable_Al[249, 0] := 526.187; fTable_Al[249, 1] := 12.2852; fTable_Al[249, 2] := 2.25125;
    fTable_Al[250, 0] := 534.698; fTable_Al[250, 1] := 12.2801; fTable_Al[250, 2] := 2.19625;
    fTable_Al[251, 0] := 543.346; fTable_Al[251, 1] := 12.2748; fTable_Al[251, 2] := 2.14277;
    fTable_Al[252, 0] := 552.134; fTable_Al[252, 1] := 12.2700; fTable_Al[252, 2] := 2.09062;
    fTable_Al[253, 0] := 561.065; fTable_Al[253, 1] := 12.2653; fTable_Al[253, 2] := 2.03805;
    fTable_Al[254, 0] := 570.139; fTable_Al[254, 1] := 12.2592; fTable_Al[254, 2] := 1.98589;
    fTable_Al[255, 0] := 579.361; fTable_Al[255, 1] := 12.2522; fTable_Al[255, 2] := 1.93406;
    fTable_Al[256, 0] := 588.732; fTable_Al[256, 1] := 12.2437; fTable_Al[256, 2] := 1.88338;
    fTable_Al[257, 0] := 598.254; fTable_Al[257, 1] := 12.2344; fTable_Al[257, 2] := 1.83389;
    fTable_Al[258, 0] := 607.930; fTable_Al[258, 1] := 12.2243; fTable_Al[258, 2] := 1.78571;
    fTable_Al[259, 0] := 617.763; fTable_Al[259, 1] := 12.2138; fTable_Al[259, 2] := 1.73879;
    fTable_Al[260, 0] := 627.755; fTable_Al[260, 1] := 12.2034; fTable_Al[260, 2] := 1.69298;
    fTable_Al[261, 0] := 637.908; fTable_Al[261, 1] := 12.1929; fTable_Al[261, 2] := 1.64704;
    fTable_Al[262, 0] := 648.226; fTable_Al[262, 1] := 12.1814; fTable_Al[262, 2] := 1.60038;
    fTable_Al[263, 0] := 658.711; fTable_Al[263, 1] := 12.1674; fTable_Al[263, 2] := 1.55377;
    fTable_Al[264, 0] := 669.365; fTable_Al[264, 1] := 12.1491; fTable_Al[264, 2] := 1.50856;
    fTable_Al[265, 0] := 680.191; fTable_Al[265, 1] := 12.1287; fTable_Al[265, 2] := 1.46882;
    fTable_Al[266, 0] := 691.193; fTable_Al[266, 1] := 12.1108; fTable_Al[266, 2] := 1.43328;
    fTable_Al[267, 0] := 702.372; fTable_Al[267, 1] := 12.0954; fTable_Al[267, 2] := 1.39941;
    fTable_Al[268, 0] := 713.733; fTable_Al[268, 1] := 12.0820; fTable_Al[268, 2] := 1.36380;
    fTable_Al[269, 0] := 725.277; fTable_Al[269, 1] := 12.0674; fTable_Al[269, 2] := 1.32737;
    fTable_Al[270, 0] := 737.008; fTable_Al[270, 1] := 12.0514; fTable_Al[270, 2] := 1.29193;
    fTable_Al[271, 0] := 748.928; fTable_Al[271, 1] := 12.0350; fTable_Al[271, 2] := 1.25742;
    fTable_Al[272, 0] := 761.042; fTable_Al[272, 1] := 12.0181; fTable_Al[272, 2] := 1.22382;
    fTable_Al[273, 0] := 773.351; fTable_Al[273, 1] := 12.0009; fTable_Al[273, 2] := 1.19100;
    fTable_Al[274, 0] := 785.859; fTable_Al[274, 1] := 11.9834; fTable_Al[274, 2] := 1.15872;
    fTable_Al[275, 0] := 798.570; fTable_Al[275, 1] := 11.9652; fTable_Al[275, 2] := 1.12705;
    fTable_Al[276, 0] := 811.486; fTable_Al[276, 1] := 11.9463; fTable_Al[276, 2] := 1.09624;
    fTable_Al[277, 0] := 824.611; fTable_Al[277, 1] := 11.9269; fTable_Al[277, 2] := 1.06625;
    fTable_Al[278, 0] := 837.949; fTable_Al[278, 1] := 11.9070; fTable_Al[278, 2] := 1.03708;
    fTable_Al[279, 0] := 851.502; fTable_Al[279, 1] := 11.8866; fTable_Al[279, 2] := 1.00870;
    fTable_Al[280, 0] := 865.274; fTable_Al[280, 1] := 11.8656; fTable_Al[280, 2] := 0.981035;
    fTable_Al[281, 0] := 879.269; fTable_Al[281, 1] := 11.8441; fTable_Al[281, 2] := 0.954065;
    fTable_Al[282, 0] := 893.491; fTable_Al[282, 1] := 11.8220; fTable_Al[282, 2] := 0.927842;
    fTable_Al[283, 0] := 907.943; fTable_Al[283, 1] := 11.7992; fTable_Al[283, 2] := 0.902346;
    fTable_Al[284, 0] := 922.628; fTable_Al[284, 1] := 11.7759; fTable_Al[284, 2] := 0.877557;
    fTable_Al[285, 0] := 937.551; fTable_Al[285, 1] := 11.7519; fTable_Al[285, 2] := 0.853321;
    fTable_Al[286, 0] := 952.715; fTable_Al[286, 1] := 11.7270; fTable_Al[286, 2] := 0.829761;
    fTable_Al[287, 0] := 968.124; fTable_Al[287, 1] := 11.7013; fTable_Al[287, 2] := 0.806859;
    fTable_Al[288, 0] := 983.783; fTable_Al[288, 1] := 11.6747; fTable_Al[288, 2] := 0.784555;
    fTable_Al[289, 0] := 999.695; fTable_Al[289, 1] := 11.6472; fTable_Al[289, 2] := 0.762967;
    fTable_Al[290, 0] := 1015.86; fTable_Al[290, 1] := 11.6184; fTable_Al[290, 2] := 0.742081;
    fTable_Al[291, 0] := 1032.29; fTable_Al[291, 1] := 11.5888; fTable_Al[291, 2] := 0.722661;
    fTable_Al[292, 0] := 1048.99; fTable_Al[292, 1] := 11.5591; fTable_Al[292, 2] := 0.703173;
    fTable_Al[293, 0] := 1065.96; fTable_Al[293, 1] := 11.5278; fTable_Al[293, 2] := 0.683588;
    fTable_Al[294, 0] := 1083.20; fTable_Al[294, 1] := 11.4947; fTable_Al[294, 2] := 0.664537;
    fTable_Al[295, 0] := 1100.72; fTable_Al[295, 1] := 11.4600; fTable_Al[295, 2] := 0.646018;
    fTable_Al[296, 0] := 1118.52; fTable_Al[296, 1] := 11.4234; fTable_Al[296, 2] := 0.628015;
    fTable_Al[297, 0] := 1136.61; fTable_Al[297, 1] := 11.3849; fTable_Al[297, 2] := 0.610519;
    fTable_Al[298, 0] := 1155; fTable_Al[298, 1] := 11.3440; fTable_Al[298, 2] := 0.593506;
    fTable_Al[299, 0] := 1173.68; fTable_Al[299, 1] := 11.3007; fTable_Al[299, 2] := 0.576965;
    fTable_Al[300, 0] := 1192.66; fTable_Al[300, 1] := 11.2544; fTable_Al[300, 2] := 0.560888;
    fTable_Al[301, 0] := 1211.95; fTable_Al[301, 1] := 11.2049; fTable_Al[301, 2] := 0.545258;
    fTable_Al[302, 0] := 1231.55; fTable_Al[302, 1] := 11.1516; fTable_Al[302, 2] := 0.530064;
    fTable_Al[303, 0] := 1251.47; fTable_Al[303, 1] := 11.0938; fTable_Al[303, 2] := 0.515441;
    fTable_Al[304, 0] := 1271.72; fTable_Al[304, 1] := 11.0310; fTable_Al[304, 2] := 0.501380;
    fTable_Al[305, 0] := 1292.29; fTable_Al[305, 1] := 10.9622; fTable_Al[305, 2] := 0.487892;
    fTable_Al[306, 0] := 1313.19; fTable_Al[306, 1] := 10.8865; fTable_Al[306, 2] := 0.474763;
    fTable_Al[307, 0] := 1334.43; fTable_Al[307, 1] := 10.8021; fTable_Al[307, 2] := 0.461987;
    fTable_Al[308, 0] := 1356.01; fTable_Al[308, 1] := 10.7069; fTable_Al[308, 2] := 0.449555;
    fTable_Al[309, 0] := 1377.94; fTable_Al[309, 1] := 10.5980; fTable_Al[309, 2] := 0.437459;
    fTable_Al[310, 0] := 1400.23; fTable_Al[310, 1] := 10.4713; fTable_Al[310, 2] := 0.425689;
    fTable_Al[311, 0] := 1422.88; fTable_Al[311, 1] := 10.3206; fTable_Al[311, 2] := 0.414239;
    fTable_Al[312, 0] := 1445.89; fTable_Al[312, 1] := 10.1361; fTable_Al[312, 2] := 0.403093;
    fTable_Al[313, 0] := 1469.28; fTable_Al[313, 1] := 9.90068; fTable_Al[313, 2] := 0.392100;
    fTable_Al[314, 0] := 1493.04; fTable_Al[314, 1] := 9.58044; fTable_Al[314, 2] := 0.381187;
    fTable_Al[315, 0] := 1517.19; fTable_Al[315, 1] := 9.09216; fTable_Al[315, 2] := 0.369680;
    fTable_Al[316, 0] := 1541.73; fTable_Al[316, 1] := 8.11537; fTable_Al[316, 2] := 0.358399;
    fTable_Al[317, 0] := 1559.50; fTable_Al[317, 1] := 1.89396; fTable_Al[317, 2] := 0.350553;
    fTable_Al[318, 0] := 1559.70; fTable_Al[318, 1] := 1.89589; fTable_Al[318, 2] := 4.16629;
    fTable_Al[319, 0] := 1566.67; fTable_Al[319, 1] := 7.10441; fTable_Al[319, 2] := 4.14105;
    fTable_Al[320, 0] := 1592.01; fTable_Al[320, 1] := 9.03572; fTable_Al[320, 2] := 4.05144;
    fTable_Al[321, 0] := 1617.76; fTable_Al[321, 1] := 9.80337; fTable_Al[321, 2] := 3.96379;
    fTable_Al[322, 0] := 1643.92; fTable_Al[322, 1] := 10.2995; fTable_Al[322, 2] := 3.87809;
    fTable_Al[323, 0] := 1670.51; fTable_Al[323, 1] := 10.6690; fTable_Al[323, 2] := 3.79420;
    fTable_Al[324, 0] := 1697.53; fTable_Al[324, 1] := 10.9642; fTable_Al[324, 2] := 3.71213;
    fTable_Al[325, 0] := 1724.99; fTable_Al[325, 1] := 11.2121; fTable_Al[325, 2] := 3.63182;
    fTable_Al[326, 0] := 1752.89; fTable_Al[326, 1] := 11.4254; fTable_Al[326, 2] := 3.54896;
    fTable_Al[327, 0] := 1781.24; fTable_Al[327, 1] := 11.6086; fTable_Al[327, 2] := 3.46653;
    fTable_Al[328, 0] := 1810.05; fTable_Al[328, 1] := 11.7695; fTable_Al[328, 2] := 3.38494;
    fTable_Al[329, 0] := 1839.32; fTable_Al[329, 1] := 11.9117; fTable_Al[329, 2] := 3.30527;
    fTable_Al[330, 0] := 1869.07; fTable_Al[330, 1] := 12.0391; fTable_Al[330, 2] := 3.22747;
    fTable_Al[331, 0] := 1899.30; fTable_Al[331, 1] := 12.1540; fTable_Al[331, 2] := 3.15148;
    fTable_Al[332, 0] := 1930.02; fTable_Al[332, 1] := 12.2583; fTable_Al[332, 2] := 3.07731;
    fTable_Al[333, 0] := 1961.24; fTable_Al[333, 1] := 12.3536; fTable_Al[333, 2] := 3.00489;
    fTable_Al[334, 0] := 1992.96; fTable_Al[334, 1] := 12.4408; fTable_Al[334, 2] := 2.93417;
    fTable_Al[335, 0] := 2025.20; fTable_Al[335, 1] := 12.5226; fTable_Al[335, 2] := 2.86696;
    fTable_Al[336, 0] := 2057.95; fTable_Al[336, 1] := 12.6001; fTable_Al[336, 2] := 2.79699;
    fTable_Al[337, 0] := 2091.24; fTable_Al[337, 1] := 12.6695; fTable_Al[337, 2] := 2.72803;
    fTable_Al[338, 0] := 2125.06; fTable_Al[338, 1] := 12.7334; fTable_Al[338, 2] := 2.66035;
    fTable_Al[339, 0] := 2159.43; fTable_Al[339, 1] := 12.7923; fTable_Al[339, 2] := 2.59405;
    fTable_Al[340, 0] := 2194.36; fTable_Al[340, 1] := 12.8467; fTable_Al[340, 2] := 2.52881;
    fTable_Al[341, 0] := 2229.85; fTable_Al[341, 1] := 12.8969; fTable_Al[341, 2] := 2.46498;
    fTable_Al[342, 0] := 2265.92; fTable_Al[342, 1] := 12.9433; fTable_Al[342, 2] := 2.40235;
    fTable_Al[343, 0] := 2302.57; fTable_Al[343, 1] := 12.9861; fTable_Al[343, 2] := 2.34101;
    fTable_Al[344, 0] := 2339.81; fTable_Al[344, 1] := 13.0257; fTable_Al[344, 2] := 2.28095;
    fTable_Al[345, 0] := 2377.66; fTable_Al[345, 1] := 13.0622; fTable_Al[345, 2] := 2.22204;
    fTable_Al[346, 0] := 2416.11; fTable_Al[346, 1] := 13.0960; fTable_Al[346, 2] := 2.16445;
    fTable_Al[347, 0] := 2455.19; fTable_Al[347, 1] := 13.1272; fTable_Al[347, 2] := 2.10810;
    fTable_Al[348, 0] := 2494.90; fTable_Al[348, 1] := 13.1560; fTable_Al[348, 2] := 2.05284;
    fTable_Al[349, 0] := 2535.26; fTable_Al[349, 1] := 13.1825; fTable_Al[349, 2] := 1.99885;
    fTable_Al[350, 0] := 2576.26; fTable_Al[350, 1] := 13.2068; fTable_Al[350, 2] := 1.94606;
    fTable_Al[351, 0] := 2617.93; fTable_Al[351, 1] := 13.2292; fTable_Al[351, 2] := 1.89447;
    fTable_Al[352, 0] := 2660.27; fTable_Al[352, 1] := 13.2498; fTable_Al[352, 2] := 1.84400;
    fTable_Al[353, 0] := 2703.30; fTable_Al[353, 1] := 13.2687; fTable_Al[353, 2] := 1.79474;
    fTable_Al[354, 0] := 2747.03; fTable_Al[354, 1] := 13.2859; fTable_Al[354, 2] := 1.74651;
    fTable_Al[355, 0] := 2791.46; fTable_Al[355, 1] := 13.3016; fTable_Al[355, 2] := 1.69945;
    fTable_Al[356, 0] := 2836.61; fTable_Al[356, 1] := 13.3159; fTable_Al[356, 2] := 1.65350;
    fTable_Al[357, 0] := 2882.49; fTable_Al[357, 1] := 13.3288; fTable_Al[357, 2] := 1.60862;
    fTable_Al[358, 0] := 2929.11; fTable_Al[358, 1] := 13.3405; fTable_Al[358, 2] := 1.56481;
    fTable_Al[359, 0] := 2976.48; fTable_Al[359, 1] := 13.3510; fTable_Al[359, 2] := 1.52204;
    fTable_Al[360, 0] := 3024.63; fTable_Al[360, 1] := 13.3604; fTable_Al[360, 2] := 1.48033;
    fTable_Al[361, 0] := 3073.55; fTable_Al[361, 1] := 13.3688; fTable_Al[361, 2] := 1.43961;
    fTable_Al[362, 0] := 3123.26; fTable_Al[362, 1] := 13.3762; fTable_Al[362, 2] := 1.39989;
    fTable_Al[363, 0] := 3173.78; fTable_Al[363, 1] := 13.3827; fTable_Al[363, 2] := 1.36116;
    fTable_Al[364, 0] := 3225.11; fTable_Al[364, 1] := 13.3883; fTable_Al[364, 2] := 1.32339;
    fTable_Al[365, 0] := 3277.27; fTable_Al[365, 1] := 13.3932; fTable_Al[365, 2] := 1.28657;
    fTable_Al[366, 0] := 3330.28; fTable_Al[366, 1] := 13.3973; fTable_Al[366, 2] := 1.25064;
    fTable_Al[367, 0] := 3384.15; fTable_Al[367, 1] := 13.4007; fTable_Al[367, 2] := 1.21564;
    fTable_Al[368, 0] := 3438.88; fTable_Al[368, 1] := 13.4034; fTable_Al[368, 2] := 1.18154;
    fTable_Al[369, 0] := 3494.50; fTable_Al[369, 1] := 13.4055; fTable_Al[369, 2] := 1.14831;
    fTable_Al[370, 0] := 3551.02; fTable_Al[370, 1] := 13.4070; fTable_Al[370, 2] := 1.11591;
    fTable_Al[371, 0] := 3608.46; fTable_Al[371, 1] := 13.4080; fTable_Al[371, 2] := 1.08436;
    fTable_Al[372, 0] := 3666.82; fTable_Al[372, 1] := 13.4085; fTable_Al[372, 2] := 1.05363;
    fTable_Al[373, 0] := 3726.13; fTable_Al[373, 1] := 13.4085; fTable_Al[373, 2] := 1.02369;
    fTable_Al[374, 0] := 3786.40; fTable_Al[374, 1] := 13.4081; fTable_Al[374, 2] := 0.994542;
    fTable_Al[375, 0] := 3847.64; fTable_Al[375, 1] := 13.4072; fTable_Al[375, 2] := 0.966167;
    fTable_Al[376, 0] := 3909.87; fTable_Al[376, 1] := 13.4060; fTable_Al[376, 2] := 0.938535;
    fTable_Al[377, 0] := 3973.11; fTable_Al[377, 1] := 13.4044; fTable_Al[377, 2] := 0.911645;
    fTable_Al[378, 0] := 4037.38; fTable_Al[378, 1] := 13.4025; fTable_Al[378, 2] := 0.885448;
    fTable_Al[379, 0] := 4102.68; fTable_Al[379, 1] := 13.4003; fTable_Al[379, 2] := 0.859966;
    fTable_Al[380, 0] := 4169.03; fTable_Al[380, 1] := 13.3978; fTable_Al[380, 2] := 0.835163;
    fTable_Al[381, 0] := 4236.46; fTable_Al[381, 1] := 13.3950; fTable_Al[381, 2] := 0.811033;
    fTable_Al[382, 0] := 4304.98; fTable_Al[382, 1] := 13.3920; fTable_Al[382, 2] := 0.787559;
    fTable_Al[383, 0] := 4374.62; fTable_Al[383, 1] := 13.3888; fTable_Al[383, 2] := 0.764708;
    fTable_Al[384, 0] := 4445.37; fTable_Al[384, 1] := 13.3853; fTable_Al[384, 2] := 0.742491;
    fTable_Al[385, 0] := 4517.27; fTable_Al[385, 1] := 13.3817; fTable_Al[385, 2] := 0.720878;
    fTable_Al[386, 0] := 4590.33; fTable_Al[386, 1] := 13.3779; fTable_Al[386, 2] := 0.699839;
    fTable_Al[387, 0] := 4664.58; fTable_Al[387, 1] := 13.3739; fTable_Al[387, 2] := 0.679399;
    fTable_Al[388, 0] := 4740.03; fTable_Al[388, 1] := 13.3698; fTable_Al[388, 2] := 0.659516;
    fTable_Al[389, 0] := 4816.69; fTable_Al[389, 1] := 13.3656; fTable_Al[389, 2] := 0.640176;
    fTable_Al[390, 0] := 4894.60; fTable_Al[390, 1] := 13.3612; fTable_Al[390, 2] := 0.621389;
    fTable_Al[391, 0] := 4973.77; fTable_Al[391, 1] := 13.3568; fTable_Al[391, 2] := 0.603106;
    fTable_Al[392, 0] := 5054.21; fTable_Al[392, 1] := 13.3522; fTable_Al[392, 2] := 0.585342;
    fTable_Al[393, 0] := 5135.96; fTable_Al[393, 1] := 13.3476; fTable_Al[393, 2] := 0.568080;
    fTable_Al[394, 0] := 5219.03; fTable_Al[394, 1] := 13.3429; fTable_Al[394, 2] := 0.551279;
    fTable_Al[395, 0] := 5303.44; fTable_Al[395, 1] := 13.3381; fTable_Al[395, 2] := 0.534968;
    fTable_Al[396, 0] := 5389.22; fTable_Al[396, 1] := 13.3332; fTable_Al[396, 2] := 0.519116;
    fTable_Al[397, 0] := 5476.39; fTable_Al[397, 1] := 13.3284; fTable_Al[397, 2] := 0.503715;
    fTable_Al[398, 0] := 5564.97; fTable_Al[398, 1] := 13.3235; fTable_Al[398, 2] := 0.488726;
    fTable_Al[399, 0] := 5654.98; fTable_Al[399, 1] := 13.3185; fTable_Al[399, 2] := 0.474187;
    fTable_Al[400, 0] := 5746.44; fTable_Al[400, 1] := 13.3135; fTable_Al[400, 2] := 0.460062;
    fTable_Al[401, 0] := 5839.39; fTable_Al[401, 1] := 13.3086; fTable_Al[401, 2] := 0.446336;
    fTable_Al[402, 0] := 5933.83; fTable_Al[402, 1] := 13.3036; fTable_Al[402, 2] := 0.433003;
    fTable_Al[403, 0] := 6029.81; fTable_Al[403, 1] := 13.2986; fTable_Al[403, 2] := 0.420026;
    fTable_Al[404, 0] := 6127.33; fTable_Al[404, 1] := 13.2936; fTable_Al[404, 2] := 0.407459;
    fTable_Al[405, 0] := 6226.44; fTable_Al[405, 1] := 13.2886; fTable_Al[405, 2] := 0.395224;
    fTable_Al[406, 0] := 6327.15; fTable_Al[406, 1] := 13.2836; fTable_Al[406, 2] := 0.383348;
    fTable_Al[407, 0] := 6429.48; fTable_Al[407, 1] := 13.2786; fTable_Al[407, 2] := 0.371815;
    fTable_Al[408, 0] := 6533.48; fTable_Al[408, 1] := 13.2737; fTable_Al[408, 2] := 0.360616;
    fTable_Al[409, 0] := 6639.15; fTable_Al[409, 1] := 13.2687; fTable_Al[409, 2] := 0.349739;
    fTable_Al[410, 0] := 6746.54; fTable_Al[410, 1] := 13.2638; fTable_Al[410, 2] := 0.339182;
    fTable_Al[411, 0] := 6855.65; fTable_Al[411, 1] := 13.2590; fTable_Al[411, 2] := 0.328927;
    fTable_Al[412, 0] := 6966.54; fTable_Al[412, 1] := 13.2541; fTable_Al[412, 2] := 0.318973;
    fTable_Al[413, 0] := 7079.22; fTable_Al[413, 1] := 13.2493; fTable_Al[413, 2] := 0.309309;
    fTable_Al[414, 0] := 7193.72; fTable_Al[414, 1] := 13.2446; fTable_Al[414, 2] := 0.299926;
    fTable_Al[415, 0] := 7310.07; fTable_Al[415, 1] := 13.2398; fTable_Al[415, 2] := 0.290817;
    fTable_Al[416, 0] := 7428.31; fTable_Al[416, 1] := 13.2352; fTable_Al[416, 2] := 0.281974;
    fTable_Al[417, 0] := 7548.45; fTable_Al[417, 1] := 13.2305; fTable_Al[417, 2] := 0.273391;
    fTable_Al[418, 0] := 7670.54; fTable_Al[418, 1] := 13.2259; fTable_Al[418, 2] := 0.265058;
    fTable_Al[419, 0] := 7794.61; fTable_Al[419, 1] := 13.2214; fTable_Al[419, 2] := 0.256972;
    fTable_Al[420, 0] := 7920.68; fTable_Al[420, 1] := 13.2169; fTable_Al[420, 2] := 0.249121;
    fTable_Al[421, 0] := 8048.79; fTable_Al[421, 1] := 13.2124; fTable_Al[421, 2] := 0.241506;
    fTable_Al[422, 0] := 8178.98; fTable_Al[422, 1] := 13.2081; fTable_Al[422, 2] := 0.234114;
    fTable_Al[423, 0] := 8311.26; fTable_Al[423, 1] := 13.2037; fTable_Al[423, 2] := 0.226938;
    fTable_Al[424, 0] := 8445.69; fTable_Al[424, 1] := 13.1994; fTable_Al[424, 2] := 0.219978;
    fTable_Al[425, 0] := 8582.29; fTable_Al[425, 1] := 13.1952; fTable_Al[425, 2] := 0.213218;
    fTable_Al[426, 0] := 8721.11; fTable_Al[426, 1] := 13.1910; fTable_Al[426, 2] := 0.206663;
    fTable_Al[427, 0] := 8862.16; fTable_Al[427, 1] := 13.1869; fTable_Al[427, 2] := 0.200304;
    fTable_Al[428, 0] := 9005.50; fTable_Al[428, 1] := 13.1829; fTable_Al[428, 2] := 0.194131;
    fTable_Al[429, 0] := 9151.16; fTable_Al[429, 1] := 13.1789; fTable_Al[429, 2] := 0.188140;
    fTable_Al[430, 0] := 9299.17; fTable_Al[430, 1] := 13.1749; fTable_Al[430, 2] := 0.182331;
    fTable_Al[431, 0] := 9449.58; fTable_Al[431, 1] := 13.1711; fTable_Al[431, 2] := 0.176693;
    fTable_Al[432, 0] := 9602.42; fTable_Al[432, 1] := 13.1672; fTable_Al[432, 2] := 0.171229;
    fTable_Al[433, 0] := 9757.73; fTable_Al[433, 1] := 13.1635; fTable_Al[433, 2] := 0.165921;
    fTable_Al[434, 0] := 9915.55; fTable_Al[434, 1] := 13.1598; fTable_Al[434, 2] := 0.160780;
    fTable_Al[435, 0] := 10075.9; fTable_Al[435, 1] := 13.1561; fTable_Al[435, 2] := 0.155788;
    fTable_Al[436, 0] := 10238.9; fTable_Al[436, 1] := 13.1526; fTable_Al[436, 2] := 0.150945;
    fTable_Al[437, 0] := 10404.5; fTable_Al[437, 1] := 13.1490; fTable_Al[437, 2] := 0.146248;
    fTable_Al[438, 0] := 10572.8; fTable_Al[438, 1] := 13.1456; fTable_Al[438, 2] := 0.141693;
    fTable_Al[439, 0] := 10743.8; fTable_Al[439, 1] := 13.1422; fTable_Al[439, 2] := 0.137274;
    fTable_Al[440, 0] := 10917.6; fTable_Al[440, 1] := 13.1388; fTable_Al[440, 2] := 0.132988;
    fTable_Al[441, 0] := 11094.2; fTable_Al[441, 1] := 13.1355; fTable_Al[441, 2] := 0.128831;
    fTable_Al[442, 0] := 11273.6; fTable_Al[442, 1] := 13.1323; fTable_Al[442, 2] := 0.124800;
    fTable_Al[443, 0] := 11455.9; fTable_Al[443, 1] := 13.1291; fTable_Al[443, 2] := 0.120890;
    fTable_Al[444, 0] := 11641.2; fTable_Al[444, 1] := 13.1260; fTable_Al[444, 2] := 0.117099;
    fTable_Al[445, 0] := 11829.5; fTable_Al[445, 1] := 13.1229; fTable_Al[445, 2] := 0.113422;
    fTable_Al[446, 0] := 12020.8; fTable_Al[446, 1] := 13.1199; fTable_Al[446, 2] := 0.109856;
    fTable_Al[447, 0] := 12215.3; fTable_Al[447, 1] := 13.1170; fTable_Al[447, 2] := 0.106398;
    fTable_Al[448, 0] := 12412.8; fTable_Al[448, 1] := 13.1141; fTable_Al[448, 2] := 0.103045;
    fTable_Al[449, 0] := 12613.6; fTable_Al[449, 1] := 13.1112; fTable_Al[449, 2] := 0.0997941;
    fTable_Al[450, 0] := 12817.6; fTable_Al[450, 1] := 13.1084; fTable_Al[450, 2] := 0.0966416;
    fTable_Al[451, 0] := 13025.0; fTable_Al[451, 1] := 13.1057; fTable_Al[451, 2] := 0.0935848;
    fTable_Al[452, 0] := 13235.6; fTable_Al[452, 1] := 13.1030; fTable_Al[452, 2] := 0.0906209;
    fTable_Al[453, 0] := 13449.7; fTable_Al[453, 1] := 13.1004; fTable_Al[453, 2] := 0.0877473;
    fTable_Al[454, 0] := 13667.2; fTable_Al[454, 1] := 13.0978; fTable_Al[454, 2] := 0.0849611;
    fTable_Al[455, 0] := 13888.3; fTable_Al[455, 1] := 13.0953; fTable_Al[455, 2] := 0.0822598;
    fTable_Al[456, 0] := 14112.9; fTable_Al[456, 1] := 13.0928; fTable_Al[456, 2] := 0.0796408;
    fTable_Al[457, 0] := 14341.2; fTable_Al[457, 1] := 13.0903; fTable_Al[457, 2] := 0.0771018;
    fTable_Al[458, 0] := 14573.1; fTable_Al[458, 1] := 13.0880; fTable_Al[458, 2] := 0.0746402;
    fTable_Al[459, 0] := 14808.9; fTable_Al[459, 1] := 13.0856; fTable_Al[459, 2] := 0.0722539;
    fTable_Al[460, 0] := 15048.4; fTable_Al[460, 1] := 13.0833; fTable_Al[460, 2] := 0.0699405;
    fTable_Al[461, 0] := 15291.8; fTable_Al[461, 1] := 13.0811; fTable_Al[461, 2] := 0.0676979;
    fTable_Al[462, 0] := 15539.1; fTable_Al[462, 1] := 13.0789; fTable_Al[462, 2] := 0.0655240;
    fTable_Al[463, 0] := 15790.4; fTable_Al[463, 1] := 13.0768; fTable_Al[463, 2] := 0.0634165;
    fTable_Al[464, 0] := 16045.8; fTable_Al[464, 1] := 13.0746; fTable_Al[464, 2] := 0.0613737;
    fTable_Al[465, 0] := 16305.4; fTable_Al[465, 1] := 13.0726; fTable_Al[465, 2] := 0.0593935;
    fTable_Al[466, 0] := 16569.1; fTable_Al[466, 1] := 13.0706; fTable_Al[466, 2] := 0.0574741;
    fTable_Al[467, 0] := 16837.1; fTable_Al[467, 1] := 13.0686; fTable_Al[467, 2] := 0.0556136;
    fTable_Al[468, 0] := 17109.4; fTable_Al[468, 1] := 13.0667; fTable_Al[468, 2] := 0.0538102;
    fTable_Al[469, 0] := 17386.1; fTable_Al[469, 1] := 13.0648; fTable_Al[469, 2] := 0.0520623;
    fTable_Al[470, 0] := 17667.4; fTable_Al[470, 1] := 13.0629; fTable_Al[470, 2] := 0.0503681;
    fTable_Al[471, 0] := 17953.1; fTable_Al[471, 1] := 13.0611; fTable_Al[471, 2] := 0.0487260;
    fTable_Al[472, 0] := 18243.5; fTable_Al[472, 1] := 13.0593; fTable_Al[472, 2] := 0.0471345;
    fTable_Al[473, 0] := 18538.6; fTable_Al[473, 1] := 13.0576; fTable_Al[473, 2] := 0.0455920;
    fTable_Al[474, 0] := 18838.4; fTable_Al[474, 1] := 13.0559; fTable_Al[474, 2] := 0.0440970;
    fTable_Al[475, 0] := 19143.1; fTable_Al[475, 1] := 13.0542; fTable_Al[475, 2] := 0.0426482;
    fTable_Al[476, 0] := 19452.7; fTable_Al[476, 1] := 13.0526; fTable_Al[476, 2] := 0.0412440;
    fTable_Al[477, 0] := 19767.4; fTable_Al[477, 1] := 13.0510; fTable_Al[477, 2] := 0.0398831;
    fTable_Al[478, 0] := 20087.1; fTable_Al[478, 1] := 13.0494; fTable_Al[478, 2] := 0.0385533;
    fTable_Al[479, 0] := 20412.0; fTable_Al[479, 1] := 13.0479; fTable_Al[479, 2] := 0.0372771;
    fTable_Al[480, 0] := 20742.1; fTable_Al[480, 1] := 13.0464; fTable_Al[480, 2] := 0.0360423;
    fTable_Al[481, 0] := 21077.6; fTable_Al[481, 1] := 13.0449; fTable_Al[481, 2] := 0.0348475;
    fTable_Al[482, 0] := 21418.5; fTable_Al[482, 1] := 13.0435; fTable_Al[482, 2] := 0.0336915;
    fTable_Al[483, 0] := 21765.0; fTable_Al[483, 1] := 13.0421; fTable_Al[483, 2] := 0.0325731;
    fTable_Al[484, 0] := 22117.0; fTable_Al[484, 1] := 13.0407; fTable_Al[484, 2] := 0.0314909;
    fTable_Al[485, 0] := 22474.7; fTable_Al[485, 1] := 13.0394; fTable_Al[485, 2] := 0.0304440;
    fTable_Al[486, 0] := 22838.2; fTable_Al[486, 1] := 13.0381; fTable_Al[486, 2] := 0.0294311;
    fTable_Al[487, 0] := 23207.6; fTable_Al[487, 1] := 13.0368; fTable_Al[487, 2] := 0.0284511;
    fTable_Al[488, 0] := 23583.0; fTable_Al[488, 1] := 13.0356; fTable_Al[488, 2] := 0.0275030;
    fTable_Al[489, 0] := 23964.4; fTable_Al[489, 1] := 13.0343; fTable_Al[489, 2] := 0.0265858;
    fTable_Al[490, 0] := 24352.0; fTable_Al[490, 1] := 13.0331; fTable_Al[490, 2] := 0.0256985;
    fTable_Al[491, 0] := 24745.9; fTable_Al[491, 1] := 13.0320; fTable_Al[491, 2] := 0.0248401;
    fTable_Al[492, 0] := 25146.2; fTable_Al[492, 1] := 13.0308; fTable_Al[492, 2] := 0.0240097;
    fTable_Al[493, 0] := 25552.9; fTable_Al[493, 1] := 13.0297; fTable_Al[493, 2] := 0.0232064;
    fTable_Al[494, 0] := 25966.2; fTable_Al[494, 1] := 13.0287; fTable_Al[494, 2] := 0.0224293;
    fTable_Al[495, 0] := 26386.1; fTable_Al[495, 1] := 13.0276; fTable_Al[495, 2] := 0.0216776;
    fTable_Al[496, 0] := 26812.9; fTable_Al[496, 1] := 13.0266; fTable_Al[496, 2] := 0.0209505;
    fTable_Al[497, 0] := 27246.6; fTable_Al[497, 1] := 13.0256; fTable_Al[497, 2] := 0.0202471;
    fTable_Al[498, 0] := 27687.3; fTable_Al[498, 1] := 13.0246; fTable_Al[498, 2] := 0.0195668;
    fTable_Al[499, 0] := 28135.1; fTable_Al[499, 1] := 13.0236; fTable_Al[499, 2] := 0.0189087;
    fTable_Al[500, 0] := 28590.2; fTable_Al[500, 1] := 13.0227; fTable_Al[500, 2] := 0.0182722;
    fTable_Al[501, 0] := 29052.6; fTable_Al[501, 1] := 13.0218; fTable_Al[501, 2] := 0.0176565;
    fTable_Al[502, 0] := 29522.5; fTable_Al[502, 1] := 13.0209; fTable_Al[502, 2] := 0.0170611;
    fTable_Al[503, 0] := 30000.0; fTable_Al[503, 1] := 13.0198; fTable_Al[503, 2] := 0.0164852;

